	// No source in this machine yet - see the header.
	_StarvedUpstream : BOOL;
	_BlockedDownstream : BOOL;
	_LowMaterial : BOOL;
	_MaterialExhausted : BOOL;

	// One flash clock for the whole indication system. The panel's button lamps
	// read it back through the module so every flashing lamp blinks in phase.
	_FlashTime : TIME := T#500MS;
	_Flash : BOOL;
	FlashTimer : TON;

	RedFlash : BOOL;
	RedSolid : BOOL;
	AmberFlash : BOOL;
	AmberSolid : BOOL;
	BlueFlash : BOOL;
	BlueSolid : BOOL;
	GreenFlash : BOOL;
	GreenSolid : BOOL;

	// Signal tower - the four lamps as driven, and the conditions behind them
	{ attribute 'TcHmiSymbol.AddSymbol' }
	HMI : ST_SignalTower_HMI;
END_VAR

// Amber solid. No source in this machine yet.
PROPERTY BlockedDownstream : BOOL
GET
BlockedDownstream := _BlockedDownstream;
END_GET
SET
_BlockedDownstream := BlockedDownstream;
END_SET
END_PROPERTY

METHOD PUBLIC CyclicLogic
VAR_INPUT
END_VAR
IF NOT _InitComplete THEN
	_InitComplete := Initialize();
	RETURN;
END_IF

// --- Flash clock ------------------------------------------------------------
// Self-retriggering TON. One clock for every flashing lamp on the machine.
FlashTimer(IN := NOT FlashTimer.Q, PT := _FlashTime);
IF FlashTimer.Q THEN
	_Flash := NOT _Flash;
END_IF

// --- Red: Abnormal Stop (flash) / Controlled Stop (solid) -------------------
RedFlash :=	(_State = Tc3_PackML_V2.E_PMLState.ePMLState_Aborting)
		OR	(_State = Tc3_PackML_V2.E_PMLState.ePMLState_Clearing)
		OR	(_State = Tc3_PackML_V2.E_PMLState.ePMLState_Aborted);

RedSolid :=	(_State = Tc3_PackML_V2.E_PMLState.ePMLState_Complete)
		OR	(_State = Tc3_PackML_V2.E_PMLState.ePMLState_Stopped)
		OR	(_State = Tc3_PackML_V2.E_PMLState.ePMLState_Stopping)
		OR	(_State = Tc3_PackML_V2.E_PMLState.ePMLState_Resetting);

// --- Amber: Starved Upstream (flash) / Blocked Downstream (solid) -----------
AmberFlash := _StarvedUpstream AND
			((_State = Tc3_PackML_V2.E_PMLState.ePMLState_Suspending)
		OR	 (_State = Tc3_PackML_V2.E_PMLState.ePMLState_Suspended));

AmberSolid := _BlockedDownstream AND
			((_State = Tc3_PackML_V2.E_PMLState.ePMLState_Suspending)
		OR	 (_State = Tc3_PackML_V2.E_PMLState.ePMLState_Suspended));

// --- Blue: Low Material (flash) / Material Exhausted (solid) ----------------
// Low Material flashes in every state EXCEPT Holding and Held, which is where
// Material Exhausted takes the lamp solid instead.
BlueFlash := _LowMaterial AND
		NOT	((_State = Tc3_PackML_V2.E_PMLState.ePMLState_Holding)
		OR	 (_State = Tc3_PackML_V2.E_PMLState.ePMLState_Held));

BlueSolid := _MaterialExhausted AND
			((_State = Tc3_PackML_V2.E_PMLState.ePMLState_Holding)
		OR	 (_State = Tc3_PackML_V2.E_PMLState.ePMLState_Held));

// --- Green: Ready to Start (flash) / Running (solid) ------------------------
GreenFlash := (_State = Tc3_PackML_V2.E_PMLState.ePMLState_Idle);

GreenSolid :=	(_State = Tc3_PackML_V2.E_PMLState.ePMLState_Starting)
			OR	(_State = Tc3_PackML_V2.E_PMLState.ePMLState_Execute)
			OR	(_State = Tc3_PackML_V2.E_PMLState.ePMLState_Completing)
			OR	(_State = Tc3_PackML_V2.E_PMLState.ePMLState_Unholding)
			OR	(_State = Tc3_PackML_V2.E_PMLState.ePMLState_Unsuspending);

// --- Drive the lamps --------------------------------------------------------
Red	:= (RedFlash	AND _Flash) OR RedSolid;
Yellow	:= (AmberFlash	AND _Flash) OR AmberSolid;
Blue	:= (BlueFlash	AND _Flash) OR BlueSolid;
Green	:= (GreenFlash	AND _Flash) OR GreenSolid;

_Busy	:= FALSE;
_Error	:= FALSE;

SUPER^.CyclicLogic();

// Device config and status only; the inherited half is bridged in
// HMICommunication. The lamps are published ALREADY BLENDED - a flashing lamp
// reads TRUE/FALSE at the flash rate - so a panel bound to these mirrors the
// real tower instead of re-deriving the state table and drifting from it.
HMI.DeviceConfig.FlashTime		:= _FlashTime;
HMI.Device.Red					:= Red;
HMI.Device.Yellow				:= Yellow;
HMI.Device.Blue					:= Blue;
HMI.Device.Green				:= Green;
HMI.Device.Flash				:= _Flash;
HMI.Device.StarvedUpstream		:= _StarvedUpstream;
HMI.Device.BlockedDownstream	:= _BlockedDownstream;
HMI.Device.LowMaterial			:= _LowMaterial;
HMI.Device.MaterialExhausted	:= _MaterialExhausted;
END_METHOD

METHOD PROTECTED HMICommunication
VAR_INPUT
END_VAR
// HMI is a published mirror of the base's own ComponentBase_HMI - carry operator
// intent in before the base looks, and its answers back out afterwards.
ComponentBase_HMI.Command := HMI.Command;

SUPER^.HMICommunication();

HMI.Config	:= ComponentBase_HMI.Config;
HMI.Status	:= ComponentBase_HMI.Status;
HMI.Command	:= ComponentBase_HMI.Command;

// A zero flash time would stop the clock dead and leave every flashing lamp
// stuck on whichever half it was in, so it is refused rather than obeyed.
IF HMI.DeviceConfig.FlashTime > T#0S THEN
	_FlashTime := HMI.DeviceConfig.FlashTime;
END_IF
END_METHOD

// The shared flash phase, so the panel's button lamps blink with the tower.
PROPERTY Flash : BOOL
GET
Flash := _Flash;
END_GET
END_PROPERTY

// Half period of the flash clock.
PROPERTY FlashTime : TIME
GET
FlashTime := _FlashTime;
END_GET
SET
_FlashTime := FlashTime;
END_SET
END_PROPERTY

METHOD PROTECTED Initialize : BOOL
VAR_INPUT
END_VAR
Initialize := SUPER^.Initialize();
END_METHOD

// Blue flashing. No source in this machine yet.
PROPERTY LowMaterial : BOOL
GET
LowMaterial := _LowMaterial;
END_GET
SET
_LowMaterial := LowMaterial;
END_SET
END_PROPERTY

// Blue solid. No source in this machine yet.
PROPERTY MaterialExhausted : BOOL
GET
MaterialExhausted := _MaterialExhausted;
END_GET
SET
_MaterialExhausted := MaterialExhausted;
END_SET
END_PROPERTY

// Amber flashing. No source in this machine yet.
PROPERTY StarvedUpstream : BOOL
GET
StarvedUpstream := _StarvedUpstream;
END_GET
SET
_StarvedUpstream := StarvedUpstream;
END_SET
END_PROPERTY

// The MACHINE's PackML state, written down by the owning module every scan.
PROPERTY State : Tc3_PackML_V2.E_PMLState
GET
State := _State;
END_GET
SET
_State := State;
END_SET
END_PROPERTY

END_FUNCTION_BLOCK

// ---- Library/POUs/F_PMLStateName.TcPOU
// The PackML state as text, for an HMI to display directly.
// IN THE PLC, NOT THE PANEL: tchmiconfig.json sets binding.symbolError to
// "Ignore", so a client-side enum conversion that fails to resolve renders an
// empty control and reports nothing, anywhere.
// Names are the Tc3_PackML_V2 members with the ePMLState_ prefix dropped.
FUNCTION F_PMLStateName : STRING(20)
VAR_INPUT
	State	: E_PMLState;
END_VAR

CASE State OF
	E_PMLState.ePMLState_Clearing:		F_PMLStateName := 'Clearing';
	E_PMLState.ePMLState_Stopped:		F_PMLStateName := 'Stopped';
	E_PMLState.ePMLState_Starting:		F_PMLStateName := 'Starting';
	E_PMLState.ePMLState_Idle:			F_PMLStateName := 'Idle';
	E_PMLState.ePMLState_Suspended:		F_PMLStateName := 'Suspended';
	E_PMLState.ePMLState_Execute:		F_PMLStateName := 'Execute';
	E_PMLState.ePMLState_Stopping:		F_PMLStateName := 'Stopping';
	E_PMLState.ePMLState_Aborting:		F_PMLStateName := 'Aborting';
	E_PMLState.ePMLState_Aborted:		F_PMLStateName := 'Aborted';
	E_PMLState.ePMLState_Holding:		F_PMLStateName := 'Holding';
	E_PMLState.ePMLState_Held:			F_PMLStateName := 'Held';
	E_PMLState.ePMLState_Unholding:		F_PMLStateName := 'Unholding';
	E_PMLState.ePMLState_Suspending:	F_PMLStateName := 'Suspending';
	E_PMLState.ePMLState_Unsuspending:	F_PMLStateName := 'Unsuspending';
	E_PMLState.ePMLState_Resetting:		F_PMLStateName := 'Resetting';
	E_PMLState.ePMLState_Completing:	F_PMLStateName := 'Completing';
	E_PMLState.ePMLState_Complete:		F_PMLStateName := 'Complete';
ELSE
	// ePMLState_Undefined, and anything a future library version adds.
	F_PMLStateName := 'Undefined';
END_CASE

END_FUNCTION

// ---- Modules/10 FG_Transport/FG_Transport.TcPOU
// FG_Transport - two level pallet conveyor, Bosch TS style, closed ring.
// Eleven stations: 5 Index, 4 Stopper, 2 Lift, plus the two main conveyors,
// which are the only thing this level owns itself.
// WireRing is the ONLY place the chain order exists - no station knows what
// follows it, which is what lets one FB serve five index units.
// Contract: _workflow/reference/transport-behaviour.md
FUNCTION_BLOCK FG_Transport EXTENDS FB_PackML_BaseModule
VAR	
	Index01			: FB_TransferIndex := (Name := 'Index01');
	Index02			: FB_TransferIndex := (Name := 'Index02');
	Index03			: FB_TransferIndex := (Name := 'Index03');
	Index04			: FB_TransferIndex := (Name := 'Index04');
	Index05			: FB_TransferIndex := (Name := 'Index05');
	Stopper01		: FB_TransferStopper := (Name := 'Stopper01');
	Stopper02		: FB_TransferStopper := (Name := 'Stopper02');
	Stopper03		: FB_TransferStopper := (Name := 'Stopper03');
	Stopper04		: FB_TransferStopper := (Name := 'Stopper04');
	Lift01			: FB_TransferLift := (Name := 'Lift01');
	Lift02			: FB_TransferLift := (Name := 'Lift02');
	Transport01		: FB_AbstractBinaryDrive := (Name := 'Transport01');
	Transport02		: FB_AbstractBinaryDrive := (Name := 'Transport02');
	
	{ attribute 'TcHmiSymbol.AddSymbol' }
	HMI : ST_BaseModule_HMI;
END_VAR

METHOD PROTECTED Aborting
VAR_INPUT
END_VAR
CASE SequenceState OF
	0:
		NoStateTasksToComplete	:= FALSE;
		Transport01.RunForward := FALSE;
		Transport01.RunBackward := FALSE;
		Transport02.RunForward := FALSE;
		Transport02.RunBackward := FALSE;
		SequenceState			:= SequenceState + 10;

	10:
		StateTasksComplete := TRUE;
END_CASE

SUPER^.Aborting();
END_METHOD

METHOD PROTECTED Clearing
VAR_INPUT
END_VAR
CASE SequenceState OF
	0:
		NoStateTasksToComplete := FALSE;
		SequenceState := SequenceState + 10;

	10:
		IF Transport01.Reset() AND Transport02.Reset() THEN
			StateTasksComplete := TRUE;
		END_IF
END_CASE

SUPER^.Clearing();
END_METHOD

METHOD PUBLIC CyclicLogic
VAR_INPUT
END_VAR
IF NOT _InitComplete THEN
	_InitComplete := Initialize();
	RETURN;
END_IF

// Ring wiring, then the state machine. There is no process image step: every
// component owns its hardware variables and is linked to a terminal channel by
// the imported Mapping_PLC.xml, not by anything in this file.
//
// The chain order lives here and nowhere else - no sub module knows which unit
// follows it. Done before the state machine so a unit sees this scan's values.
WireRing();

// Components get no PackML state callbacks, so the owning module removes every run
// request outside the states entitled to drive them.
// TWO STATES DRIVE THE CONVEYORS: Execute, and Resetting - which runs them to
// accumulate loose pallets against the blocking stoppers.
// THIS GUARD RUNS BEFORE SUPER^.CyclicLogic(), so it does not merely veto the
// output for a scan - it ERASES the request the state method set on the previous
// scan. A state left out of this condition cannot move a conveyor at all,
// however plainly its own code commands one.
IF (_CurrentState <> E_PMLState.ePMLState_Execute)
	AND (_CurrentState <> E_PMLState.ePMLState_Resetting) THEN
	Transport01.RunForward := FALSE;
	Transport01.RunBackward := FALSE;
	Transport02.RunForward := FALSE;
	Transport02.RunBackward := FALSE;
END_IF

SUPER^.CyclicLogic();

PublishStatus();
END_METHOD

METHOD PROTECTED Execute
VAR_INPUT
END_VAR
// The stations sequence themselves - SUPER^.Execute() drives all eleven sub
// modules' Execute methods. This level only owns what belongs to no station:
// the two main conveyors.
//
// There is no step chain here and no completion. A transport ring runs until it
// is stopped, so Execute never calls Complete.

CASE _CurrentMode OF

	//============================= PRODUCTION =================================
	E_PMLUnitMode.ePMLUnitMode_Production:		
		Transport01.RunBackward := TRUE;
		Transport02.RunBackward := TRUE;
		Transport01.RunForward  := FALSE;
		Transport02.RunForward  := FALSE;

	//======================= MAINTENANCE & MANUAL =============================
	E_PMLUnitMode.ePMLUnitMode_Maintenance, E_PMLUnitMode.ePMLUnitMode_Manual:
		// Nothing to do at this level. Each drive honours its own
		// HMI.DeviceCommand struct in these modes - see
		// FB_AbstractBinaryDrive.HMICommunication - so a panel talks to the
		// device it is pointing at rather than through a group GVL. The eleven
		// stations' cylinders do the same through their SPT SolenoidHMI structs.
		;
END_CASE

SUPER^.Execute();
END_METHOD

METHOD PROTECTED HMICommunication
VAR_INPUT
END_VAR
// The command half of the HMI bridge; PublishStatus is the status half.
//
// Without this, the group's published Command block is decoration: the base reads
// its own PackMLBaseModule_HMI.Command and never looks at ours, so a mode or state
// button on the FG_Transport tile would write into a struct nothing consumes.
// It has to happen here because the base calls this method immediately before
// ModeControl() and StateControl().
PackMLBaseModule_HMI.Command := HMI.Command;

SUPER^.HMICommunication();

// The base clears a latch by writing back the value it acted on.
HMI.Command := PackMLBaseModule_HMI.Command;
END_METHOD

METHOD PROTECTED Initialize : BOOL;
VAR
END_VAR
Initialize := FALSE;

CASE DescendantSequenceState OF
	0:
		// HMI.Config.Name is NOT set here. The SPT base writes Config.Name from
		// _Name every scan in its own HMICommunication, and PublishStatus copies
		// the whole Config across - setting it here would be a second author for
		// one field and the first to drift.

		// Eleven station submodules plus two drive components. Forgetting one is
		// silent: its cyclic framework logic would simply never be called.
		RegisterSubmodule(Index01);
		RegisterSubmodule(Index02);
		RegisterSubmodule(Index03);
		RegisterSubmodule(Index04);
		RegisterSubmodule(Index05);
		RegisterSubmodule(Stopper01);
		RegisterSubmodule(Stopper02);
		RegisterSubmodule(Stopper03);
		RegisterSubmodule(Stopper04);
		RegisterSubmodule(Lift01);
		RegisterSubmodule(Lift02);
		RegisterComponent(Transport01);
		RegisterComponent(Transport02);

		// Devices that belong to the group rather than to a station.
		_LogModeChanges		:= FALSE;
		_LogStateChanges	:= TRUE;
		DescendantSequenceState := DescendantSequenceState + 10;

	10:
		// Lift01 raises: it loads at the retracted (lower) end.
		// Lift02 lowers: the mirror image. This one parameter is the entire
		// difference between the two instances.
		Lift01.ReverseDirection := FALSE;
		Lift02.ReverseDirection := TRUE;

		DescendantSequenceState := DescendantSequenceState + 10;

	20:
		IF SUPER^.Initialize() THEN
			DescendantSequenceState := DescendantSequenceState + 10;
		END_IF

	30:
		Initialize := TRUE;
END_CASE
END_METHOD

// TRUE while index unit <Index> is holding a pallet stopped and lifted, waiting
// for its functional group to run. The Machine module polls this and turns it
// into a Start command on the matching group.
//
// A method rather than five properties so the caller can loop 1..5.
METHOD PUBLIC IsIndexReadyForOperation : BOOL
VAR_INPUT
	Index : INT;	// 1..5
END_VAR
CASE Index OF
	1:	IsIndexReadyForOperation := Index01.ReadyForOperation;
	2:	IsIndexReadyForOperation := Index02.ReadyForOperation;
	3:	IsIndexReadyForOperation := Index03.ReadyForOperation;
	4:	IsIndexReadyForOperation := Index04.ReadyForOperation;
	5:	IsIndexReadyForOperation := Index05.ReadyForOperation;
ELSE
	IsIndexReadyForOperation := FALSE;
END_CASE
END_METHOD

ACTION PublishStatus:
// The status half of the HMI bridge; HMICommunication is the command half.
//
// Called from CyclicLogic AFTER SUPER^.CyclicLogic(), so everything below is this
// scan's value. The three fields this action used to set by hand - Mode, State and
// the step index - were the only three that were ever current; Busy, Error,
// ErrorID and HMIControlAvailable stayed at zero because nothing wrote them.
// Copying the base's struct wholesale fixes that and cannot drift.
HMI.Config		:= PackMLBaseModule_HMI.Config;
HMI.Status		:= PackMLBaseModule_HMI.Status;

HMI.StateName			:= F_PMLStateName(_CurrentState);
HMI.Sequence.StepIndex	:= SequenceState;
END_ACTION

METHOD PROTECTED Resetting
VAR_INPUT
END_VAR
// Every station homes itself through its own Resetting, reached by SUPER^.
// This level owns what belongs to no station: the two main conveyors.
// THE CONVEYORS RUN DURING THE RESET, in the production direction. Safe because
// nothing opens: a stopper blocks and is never released, an index blocks before
// lowering. Loose pallets accumulate against the blocking stoppers where a detect
// sensor can see them. It is also what lets a lift hand on a pallet it was
// carrying when it was interrupted, instead of pushing it onto a dead belt.

CASE SequenceState OF
	0:
		NoStateTasksToComplete	:= FALSE;
		Transport01.RunBackward := TRUE;
		Transport02.RunBackward := TRUE;
		Transport01.RunForward  := FALSE;
		Transport02.RunForward  := FALSE;
		SequenceState			:= SequenceState + 10;

	10:
		// The state does not end here: SUPER^ holds it open until all eleven stations
		// have finished their own Resetting, each ending with a fixed accumulation
		// wait, so the belts run for the whole settling period.
		// THE ACCUMULATION IS THE RESET. Once it has settled, every station's state is
		// simply what its sensor says - which is why nothing here waits on an event
		// that might never arrive.
		StateTasksComplete := TRUE;
END_CASE

SUPER^.Resetting();
END_METHOD

// Reports back to index unit <Index> that its functional group has finished, so
// the pallet may be lowered and released. Written by the Machine module.
//
// The index unit clears the flag itself once it has seen it - the group never has
// to reset anything, which is the contract the twin's SIL establishes.
METHOD PUBLIC SetIndexOperationDone
VAR_INPUT
	Index	: INT;		// 1..5
	Value	: BOOL;
END_VAR
CASE Index OF
	1:	Index01.OperationDone := Value;
	2:	Index02.OperationDone := Value;
	3:	Index03.OperationDone := Value;
	4:	Index04.OperationDone := Value;
	5:	Index05.OperationDone := Value;
END_CASE
END_METHOD

METHOD PROTECTED Stopping
VAR_INPUT
END_VAR
CASE SequenceState OF
	0:
		NoStateTasksToComplete	:= FALSE;
		// The drives are components: they have no state methods of their own, so
		// nothing here reaches them through SUPER^. The guard in CyclicLogic is
		// what stops them, and Stopping is not one of the states it exempts.
		SequenceState			:= SequenceState + 10;

	10:
		StateTasksComplete := TRUE;
END_CASE

SUPER^.Stopping();
END_METHOD

ACTION WireRing:
// The chain, exactly as probed from the scene. This is the only place the order
// is written down; no station knows what follows it, which is what lets one FB
// serve five index units.
//
//   Lift01 -> Stopper03 -> Index01 -> Index02 -> Index03 -> Index04 -> Index05
//          -> Stopper04 -> Lift02 -> Stopper01 -> Stopper02 -> Lift01
//
// THE WIRING IS THE AUTHORITY. Two authored Role entries in the twin name the
// wrong successor - both skip the intervening stopper.

// --- Successor readiness: nobody releases into a station that cannot take it ---
//
// ONE CHANNEL, VALID IN EVERY STATE. CanAccept is a derived property - cylinder
// position, detect sensor, transfer latch, no outstanding fault - so it answers
// the same question during Resetting as during Execute. That is what lets a lift's
// reset recovery hand its pallet over on the ordinary contract instead of needing
// a second, reset-only channel wired alongside this one.
Lift01.NextCanAccept	:= Stopper03.CanAccept;
Stopper03.NextCanAccept	:= Index01.CanAccept;
Index01.NextCanAccept	:= Index02.CanAccept;
Index02.NextCanAccept	:= Index03.CanAccept;
Index03.NextCanAccept	:= Index04.CanAccept;
Index04.NextCanAccept	:= Index05.CanAccept;
Index05.NextCanAccept	:= Stopper04.CanAccept;
Stopper04.NextCanAccept	:= Lift02.CanAccept;
Lift02.NextCanAccept	:= Stopper01.CanAccept;
Stopper01.NextCanAccept	:= Stopper02.CanAccept;
Stopper02.NextCanAccept	:= Lift01.CanAccept;

// --- Payload announcements ---------------------------------------------------
// Only a lift acts on being told a pallet is coming: it reverses its belt to draw
// the pallet aboard. Every other station picks a pallet up on its own detect
// sensor, so the announcement would be inert and is not wired.
//
// A lift is a pulling station; the units it feeds are pushing stations. That
// asymmetry is deliberate, not an oversight - see interfaces.md.
Lift01.PayloadIncoming := Stopper02.SendToNext;
Lift02.PayloadIncoming := Stopper04.SendToNext;
END_ACTION

END_FUNCTION_BLOCK

// ---- Modules/10 FG_Transport/FB_TransferIndex.TcPOU
// Index unit - stops a pallet, lifts it clear, runs its functional group,
// then releases. Five instances; the ring wiring decides which is which.
// CanAccept/Occupied are GETTERS, never stored: a remembered readiness flag
// maintained inside Execute is stale in every other state.
// Contract: _workflow/reference/transport-behaviour.md
FUNCTION_BLOCK FB_TransferIndex EXTENDS FB_PackML_BaseModule
VAR
	// --- Components ---------------------------------------------------------
	{ attribute 'TcHmiSymbol.AddSymbol' }
	B_Detect		: FB_DigitalSensor;
	{ attribute 'TcHmiSymbol.AddSymbol' }
	B_Exit			: FB_DigitalSensor;
	{ attribute 'TcHmiSymbol.AddSymbol' }
	Y_Lift			: FB_DoubleSolenoidFeedback;
	{ attribute 'TcHmiSymbol.AddSymbol' }
	Y_Stopper		: FB_SingleSolenoidFeedback;


	// --- Ring handshake -----------------------------------------------------
	// THE INTERFACE IS DERIVED, NOT ASSIGNED. CanAccept and Occupied are getters,
	// correct in every PackML state and mode. There is no _Ready to go stale.
	// _Transferring is the ONE piece of memory: a payload is crossing right now.
	// Set on commit to release, cleared by a B_Exit EDGE in CyclicLogic so it
	// happens in every state.
	_Transferring	: BOOL;
	// Edge detector for the clearing rule. A LEVEL cannot be used: B_Exit may still
	// be made by the previous pallet at the moment this unit commits to the next
	// release, which would clear the latch instantly. The rising edge after the
	// commit is unambiguous, and unlike a cylinder position it is not erased by
	// Stopping or Aborting.
	ExitEdge		: R_TRIG;
	// The successor can physically accept a pallet. Supplied by the parent.
	_NextCanAccept	: BOOL;

	// --- Functional group handshake -----------------------------------------
	// The group is a sibling equipment module, so the Machine module brokers this:
	// it reads ReadyForOperation, commands the group, and writes OperationDone
	// back. This unit never names a functional group.
	_ReadyForOperation	: BOOL;		// pallet is stopped and lifted - run your operation
	_OperationDone		: BOOL;		// the group reports finished

	// The group is not available: it is switched out, or it does not exist yet.
	// The pallet is still stopped, lifted and fixed exactly as always - only the
	// request to run is skipped, so the station is passed rather than skipped and
	// the ring keeps its timing. Routed in by the Machine module, same as the rest.

	// --- Diagnostics --------------------------------------------------------
	// 0 none  1 no home  2 lift did not raise  3 group did not finish
	// 4 lift did not lower  5 no release  6 pallet never reached the exit sensor
	_FaultCode		: DINT;

	// --- Parameters, set by the parent in Initialize ------------------------
	_BlockTime		: TIME := T#2S;
	_LiftTime		: TIME := T#3S;
	_OperationTime	: TIME := T#60S;	// how long a station may take
	_ReleaseTime	: TIME := T#2S;
	_ClearTime		: TIME := T#10S;
	// How long a reset lets the line settle once this unit is blocking and lowered.
	// The group runs the main conveyors throughout, so pallets travel up against the
	// blocking stoppers and accumulate where a detect sensor can see them.
	_AccumulateTime	: TIME := T#5S;

	// --- HMI ----------------------------------------------------------------
	// One struct for the whole tile, extending the SPT module interface. The
	// inherited half is bridged to the base's own PackMLBaseModule_HMI in two
	// places: HMICommunication pushes Command in before the base acts on it,
	// PublishHMI copies Config and Status back out after. The Station half is this
	// block's own and is filled by PublishHMI alone.
	{ attribute 'TcHmiSymbol.AddSymbol' }
	HMI	: ST_TransferIndex_HMI;
END_VAR

METHOD PROTECTED Aborting
VAR_INPUT
END_VAR
CASE SequenceState OF
	0:
		NoStateTasksToComplete	:= FALSE;
		// Block, and withdraw the request to the station. The lift is left where
		// it is on purpose - dropping a pallet that a station still has hold of
		// is worse than leaving it raised. An abort is immediate by definition, so
		// unlike Resetting it does not wait for a crossing to finish.
		//
		// Nothing else is cleared: the interface is derived, and _Transferring is
		// cleared by B_Exit whenever the pallet actually gets there.
		Y_Stopper.Retract();
		_ReadyForOperation	:= FALSE;
		SequenceState		:= SequenceState + 10;

	10:
		StateTasksComplete := TRUE;
END_CASE

SUPER^.Aborting();
END_METHOD

METHOD PROTECTED Clearing
VAR_INPUT
END_VAR
CASE SequenceState OF
	0:
		NoStateTasksToComplete := FALSE;
		_FaultCode := 0;
		SequenceState := SequenceState + 10;

	10:	// Clear latched component alarms - the lift's travel timeout latches.
		IF Y_Lift.Reset()
			AND Y_Stopper.Reset()
			AND B_Detect.Reset()
			AND B_Exit.Reset() THEN
			SequenceState := SequenceState + 10;
		END_IF

	20:
		StateTasksComplete := TRUE;
END_CASE

SUPER^.Clearing();
END_METHOD

METHOD PUBLIC CyclicLogic
VAR_INPUT
END_VAR
IF NOT _InitComplete THEN
	_InitComplete := Initialize();
	RETURN;
END_IF

// Nothing to copy: every component is linked to its terminal at the instance
// declaration in FG_Transport.

// THE TRANSFER LATCH IS CLEARED BY THE SENSOR, IN EVERY STATE - not in the
// Execute step that starts the release. A pallet that finishes crossing while
// the machine is stopped or resetting has still finished crossing.
//
// THE WITNESS MUST BE A SENSOR EDGE. Qualifying it with Y_Stopper.Extended
// deadlocked the machine: Stopping and Aborting retract the cylinder immediately,
// destroying the very witness the rule depended on. A rising edge is specific to
// THIS crossing and no state change can erase it.
ExitEdge(CLK := B_Exit.Active);
IF _Transferring AND ExitEdge.Q THEN
	_Transferring := FALSE;
END_IF

SUPER^.CyclicLogic();

// After the base, so the published struct carries this scan's state and
// this scan's HMI permission rather than last scan's.
PublishHMI();
END_METHOD

METHOD PROTECTED Execute
VAR_INPUT
END_VAR
VAR_INST
	HomeTimer		: TON;
	LiftUpTimer		: TON;
	OperationTimer	: TON;
	LiftDownTimer	: TON;
	ReleaseTimer	: TON;
	ClearTimer		: TON;
END_VAR
// The ring runs continuously, so this state loops instead of completing.

CASE _CurrentMode OF

	//============================= PRODUCTION =================================
	E_PMLUnitMode.ePMLUnitMode_Production:

		CASE SequenceState OF
			0:	// Home: blocking, lift down, nothing outstanding. The handshake
				// interface is derived and needs nothing cleared here; only the
				// group request, which is this unit's own bookkeeping.
				NoStateTasksToComplete	:= FALSE;
				Y_Stopper.Retract();
				Y_Lift.Retract();
				_ReadyForOperation	:= FALSE;
				_OperationDone		:= FALSE;
				SequenceState		:= SequenceState + 10;

			10:	// Blocking position comes from the real switch; the lift has a
				// genuine feedback component and reports its own position.
				// CanAccept becomes TRUE by itself once both are home and the
				// detect sensor is clear - this unit never publishes readiness, so
				// there is no window in which it advertises it over a pallet.
				IF Y_Stopper.Retracted AND Y_Lift.Retracted THEN
					SequenceState	:= SequenceState + 10;
				ELSIF HomeTimer.Q THEN
					_FaultCode := 1;
					ChangeState(E_PMLCommand.ePMLCommand_Hold);
				END_IF

			20:	// Idle and empty - the normal resting condition
				IF B_Detect.Active THEN
					SequenceState	:= SequenceState + 10;
				END_IF

			30:	// Invariant 1 - lift the pallet clear while the stopper still
				// holds it, and only then let the station run.
				Y_Lift.Extend();
				IF Y_Lift.Extended THEN
					SequenceState	:= SequenceState + 10;
				ELSIF LiftUpTimer.Q THEN
					_FaultCode := 2;
					ChangeState(E_PMLCommand.ePMLCommand_Hold);
				END_IF

			40:	// Ask the group to run and wait for it. The Machine module
				// brokers both halves; this unit clears the done flag itself, so
				// the group never has to reset anything.
				//
				// A group that is not implemented is handled by the broker, which
				// answers SetIndexOperationDone immediately - see
				// Machine.BrokerIndexHandshakes. This unit neither knows nor cares
				// which groups exist.
				_ReadyForOperation := TRUE;
				IF _OperationDone THEN
					_OperationDone		:= FALSE;
					_ReadyForOperation	:= FALSE;
					SequenceState		:= SequenceState + 10;
				ELSIF OperationTimer.Q THEN
					_FaultCode := 3;
					ChangeState(E_PMLCommand.ePMLCommand_Hold);
				END_IF

			50:	// Invariant 2 - the operation is complete, so the lift may drop
				Y_Lift.Retract();
				IF Y_Lift.Retracted THEN
					SequenceState := SequenceState + 10;
				ELSIF LiftDownTimer.Q THEN
					_FaultCode := 4;
					ChangeState(E_PMLCommand.ePMLCommand_Hold);
				END_IF

			60:	// Invariant 3 - the successor can physically accept before release
				IF _NextCanAccept THEN
					// The crossing starts here; cleared by B_Exit in CyclicLogic.
					_Transferring	:= TRUE;
					SequenceState	:= SequenceState + 10;
				END_IF

			70:	// Release
				Y_Stopper.Extend();
				IF Y_Stopper.Extended THEN
					SequenceState := SequenceState + 10;
				ELSIF ReleaseTimer.Q THEN
					_FaultCode := 5;
					ChangeState(E_PMLCommand.ePMLCommand_Hold);
				END_IF

			80:	// Confirm the pallet actually left
				IF B_Exit.Active THEN
					SequenceState := 0;
				ELSIF ClearTimer.Q THEN
					_FaultCode := 6;
					ChangeState(E_PMLCommand.ePMLCommand_Hold);
				END_IF
		END_CASE

	//======================= MAINTENANCE & MANUAL =============================
	E_PMLUnitMode.ePMLUnitMode_Maintenance, E_PMLUnitMode.ePMLUnitMode_Manual:
		// Both cylinders are SPT components and honour their own SolenoidHMI
		// structs whenever the mode grants HMI control. The handshake interface is
		// derived from the sensors, so it keeps telling the truth while an operator
		// moves pallets by hand; only the group request is withdrawn.
		_ReadyForOperation	:= FALSE;
END_CASE

SUPER^.Execute();

HomeTimer(		IN := (SequenceState = 10),							PT := _BlockTime);
LiftUpTimer(	IN := (SequenceState = 30),							PT := _LiftTime);
OperationTimer(	IN := (SequenceState = 40),							PT := _OperationTime);
LiftDownTimer(	IN := (SequenceState = 50),							PT := _LiftTime);
ReleaseTimer(	IN := (SequenceState = 70),							PT := _ReleaseTime);
ClearTimer(		IN := (SequenceState = 80),							PT := _ClearTime);
END_METHOD

// 0 none  1 no home  2 lift did not raise  3 group did not finish
// 4 lift did not lower  5 no release  6 pallet never reached the exit sensor
PROPERTY FaultCode : DINT
GET
FaultCode := _FaultCode;
END_GET
END_PROPERTY

METHOD PROTECTED HMICommunication
VAR_INPUT
END_VAR
// The command half of the HMI bridge. The status half is PublishHMI.
// MUST be in this method, not in PublishHMI. The base calls it immediately before
// ModeControl() and StateControl(), and reads its OWN PackMLBaseModule_HMI.Command,
// never ours. A command written after SUPER^.CyclicLogic() returns is a full scan
// too late, every time.
PackMLBaseModule_HMI.Command := HMI.Command;

SUPER^.HMICommunication();

// The base clears a command latch by writing the value it acted on back into
// Command.Mode / Command.State. Carry that back out so the panel sees its request
// consumed rather than re-issuing it on the next scan.
HMI.Command := PackMLBaseModule_HMI.Command;
END_METHOD

METHOD PROTECTED Initialize : BOOL;
VAR
END_VAR
Initialize := FALSE;

CASE DescendantSequenceState OF
	0:
		RegisterComponent(B_Detect);
		RegisterComponent(B_Exit);
		RegisterComponent(Y_Lift);
		RegisterComponent(Y_Stopper);

		_LogModeChanges		:= FALSE;
		_LogStateChanges	:= FALSE;
		DescendantSequenceState := DescendantSequenceState + 10;

	10:
		// Travel timeouts in ms (LREAL). The lift has real feedback so these
		// alarm on a jam; the stopper is open loop and these only bound the move.
		Y_Lift.ExtendTime		:= 3000.0;
		Y_Lift.RetractTime		:= 3000.0;
		Y_Stopper.ExtendTime	:= 2000.0;
		Y_Stopper.RetractTime	:= 2000.0;
		DescendantSequenceState := DescendantSequenceState + 10;

	20:
		IF SUPER^.Initialize() THEN
			DescendantSequenceState := DescendantSequenceState + 10;
		END_IF

	30:
		Initialize := TRUE;
END_CASE
END_METHOD

// The successor's CanAccept, wired in by the parent.
PROPERTY NextCanAccept : BOOL
SET
_NextCanAccept := NextCanAccept;
END_SET
END_PROPERTY

// This station is physically holding or handling a pallet.
//
// Derived, like CanAccept: the detect sensor, or a crossing that has been committed
// to and not yet confirmed finished. There is no remembered occupancy behind it, so
// there is nothing for a state change or a program download to falsify.
PROPERTY Occupied : BOOL
GET
Occupied := B_Detect.Active OR _Transferring;
END_GET
END_PROPERTY

// Written TRUE by the Machine module when this unit's functional group reports
// its operation complete. This unit clears it again itself.
PROPERTY OperationDone : BOOL
SET
_OperationDone := OperationDone;
END_SET
END_PROPERTY

ACTION PublishHMI:
// Everything an operator tile needs from this unit, in one struct.
//
// Called from CyclicLogic AFTER SUPER^.CyclicLogic(), so _CurrentState and the
// base's HMIControlAvailable are this scan's values and not last scan's.

// --- Inherited half ---------------------------------------------------------
// Straight copies of the struct the SPT base maintains. Nothing is recomputed -
// a second calculation would be a second answer.
// HMIControlAvailable is the gate for every jog button on the tile, and only
// ePMLUnitMode_Manual grants it. Bind button enablement to THIS, not to a
// group-level flag computed as Manual OR Maintenance, which over-reports.
HMI.Config		:= PackMLBaseModule_HMI.Config;
HMI.Status		:= PackMLBaseModule_HMI.Status;

HMI.StateName			:= F_PMLStateName(_CurrentState);
HMI.Sequence.StepIndex	:= SequenceState;

// --- Ring handshake ---------------------------------------------------------
// The derived properties, not backing variables - the tile shows what the machine
// physically is, which is the same thing the neighbouring stations act on. The
// struct field names are unchanged so the existing panel bindings still resolve.
HMI.Station.Ready					:= CanAccept;
HMI.Station.Occupied				:= Occupied;
HMI.Station.NextReady				:= _NextCanAccept;
HMI.Station.SendToNext				:= SendToNext;

// --- Functional group handshake ---------------------------------------------
HMI.Station.ReadyForOperation		:= _ReadyForOperation;
HMI.Station.OperationDone			:= _OperationDone;

// --- Diagnostics ------------------------------------------------------------
HMI.Station.FaultCode				:= _FaultCode;
END_ACTION

// This station can physically take a pallet right now. The predecessor gates its
// release on this, and it is the whole of the readiness contract.
//
// DERIVED, NOT ASSIGNED. Computed from both cylinder limit switches, the detect
// sensor and the transfer latch, so it is correct in every PackML state and every
// mode. The old _Ready was written only inside the Execute step chain, which made
// it stale or FALSE everywhere else.
PROPERTY CanAccept : BOOL
GET
CanAccept := Y_Stopper.Retracted
	AND Y_Lift.Retracted
	AND NOT B_Detect.Active
	AND NOT _Transferring
	AND (_FaultCode = 0);
END_GET
END_PROPERTY

// The pallet is stopped and lifted. The Machine module turns this into a Start
// command on the matching functional group.
PROPERTY ReadyForOperation : BOOL
GET
ReadyForOperation := _ReadyForOperation;
END_GET
END_PROPERTY

METHOD PROTECTED Resetting
VAR_INPUT
END_VAR
VAR_INST
	ResetBlockTimer	: TON;
	ResetLiftTimer	: TON;
	AccumulateTimer	: TON;
END_VAR
// A RESET RE-ESTABLISHES WHERE THE PALLETS ARE.
// Block, drop the lift, then wait for the line to settle. The group runs the main
// conveyors throughout a reset, so whatever was moving accumulates against the
// blocking stoppers; after that each station's state is what its sensor says.
//
// A FIXED WAIT, NOT AN EVENT. Waiting for the in-flight pallet to clear B_Exit
// deadlocked: Stopping had already retracted the cylinder the clearing rule
// needed. A RESET MUST ALWAYS TERMINATE - nothing in it may wait on an event that
// might not arrive.

CASE SequenceState OF
	0:
		NoStateTasksToComplete	:= FALSE;
		Y_Stopper.Retract();
		_ReadyForOperation	:= FALSE;
		_OperationDone		:= FALSE;
		// The routed inputs are not cleared here: they are rewritten every scan by the
		// Machine, and a reset is not the operator changing their mind about it.
		SequenceState		:= SequenceState + 10;

	10:	// Drop the lift only once the stopper is confirmed blocking
		IF Y_Stopper.Retracted THEN
			SequenceState := SequenceState + 10;
		ELSIF ResetBlockTimer.Q THEN
			_FaultCode := 1;
			ChangeState(E_PMLCommand.ePMLCommand_Hold);
		END_IF

	20:
		Y_Lift.Retract();
		IF Y_Lift.Retracted THEN
			SequenceState := SequenceState + 10;
		ELSIF ResetLiftTimer.Q THEN
			_FaultCode := 4;
			ChangeState(E_PMLCommand.ePMLCommand_Hold);
		END_IF

	30:	// Accumulation. When it expires the pallets have settled, so any crossing
		// this unit had outstanding is over by definition. Clearing the latch here
		// is the reset re-establishing state rather than inheriting a crossing whose
		// sensor edge was missed while the machine was stopped.
		IF AccumulateTimer.Q THEN
			_Transferring	:= FALSE;
			SequenceState	:= SequenceState + 10;
		END_IF

	40:
		StateTasksComplete := TRUE;
END_CASE

SUPER^.Resetting();

ResetBlockTimer(IN := (SequenceState = 10),							PT := _BlockTime);
ResetLiftTimer(	IN := (SequenceState = 20),							PT := _LiftTime);
AccumulateTimer(IN := (SequenceState = 30),							PT := _AccumulateTime);
END_METHOD

// This unit is handing a pallet over right now; only a lift acts on it.
//
// This is the transfer latch itself, not a second flag that shadows it. Handing
// over and being mid-crossing are the same fact, so keeping them as one variable
// means they cannot disagree. Cleared by B_Exit.
PROPERTY SendToNext : BOOL
GET
SendToNext := _Transferring;
END_GET
END_PROPERTY

METHOD PROTECTED Stopping
VAR_INPUT
END_VAR
// A controlled stop blocks and withdraws the station request, but leaves the
// lift alone so a part being worked on is not dropped mid-operation.

CASE SequenceState OF
	0:
		NoStateTasksToComplete	:= FALSE;
		// Block and withdraw the station request. Nothing to clear - see Aborting.
		Y_Stopper.Retract();
		_ReadyForOperation	:= FALSE;
		SequenceState		:= SequenceState + 10;

	10:
		StateTasksComplete := TRUE;
END_CASE

SUPER^.Stopping();
END_METHOD

END_FUNCTION_BLOCK

// ---- Modules/10 FG_Transport/FB_TransferStopper.TcPOU
// Accumulation stopper - one pallet, held until the next station is free.
// RETRACTED (min) HOLDS THE PALLET; EXTENDING (max) RELEASES IT. Nine authored
// Function entries in the twin once said the opposite.
// CanAccept/Occupied are GETTERS, never stored.
// Contract: _workflow/reference/transport-behaviour.md
FUNCTION_BLOCK FB_TransferStopper EXTENDS FB_PackML_BaseModule
VAR
	// --- Components ---------------------------------------------------------
	{ attribute 'TcHmiSymbol.AddSymbol' }
	B_Detect		: FB_DigitalSensor;
	{ attribute 'TcHmiSymbol.AddSymbol' }
	B_Exit			: FB_DigitalSensor;
	{ attribute 'TcHmiSymbol.AddSymbol' }
	Y_Stopper		: FB_SingleSolenoidFeedback;


	// --- Ring handshake -----------------------------------------------------
	// THE INTERFACE IS DERIVED, NOT ASSIGNED. CanAccept and Occupied are getters,
	// correct in every PackML state and mode. There is no _Ready to go stale.
	// _Transferring is the ONE piece of memory: a payload is crossing right now.
	// Set on commit to release, cleared by a B_Exit EDGE in CyclicLogic so it
	// happens in every state. A plain BOOL initialising FALSE is the point - a
	// stale FALSE is corrected by B_Detect on the next scan.
	_Transferring	: BOOL;
	// Edge detector for the clearing rule. A LEVEL cannot be used: B_Exit may still
	// be made by the previous pallet at the moment this unit commits to the next
	// release, which would clear the latch instantly. The rising edge after the
	// commit is unambiguous, and unlike a cylinder position or a drive command it
	// is not erased by Stopping or Aborting.
	ExitEdge		: R_TRIG;
	// The successor can physically accept a pallet. Supplied by the parent.
	_NextCanAccept	: BOOL;

	// --- Diagnostics --------------------------------------------------------

	// Module level fault. The SPT components raise their own alarms through the
	// event logger; these codes cover the sequence timeouts, which belong to the
	// unit rather than to any one device. Published for the HMI.
	// 0 none  1 no block  2 no release  3 pallet never reached the exit sensor
	_FaultCode		: DINT;

	// --- Parameters, set by the parent in Initialize ------------------------
	_BlockTime		: TIME := T#2S;		// stopper travel to the blocking position
	_ReleaseTime	: TIME := T#2S;		// stopper travel to the release position
	_ClearTime		: TIME := T#10S;	// pallet to reach the exit sensor once released
	// How long a reset lets the line settle once this unit is blocking. The group
	// runs the main conveyors throughout, so pallets travel up against the blocking
	// stoppers and accumulate where a detect sensor can see them.
	_AccumulateTime	: TIME := T#5S;

	// --- HMI ----------------------------------------------------------------
	// One struct for the whole tile, extending the SPT module interface. The
	// inherited half is bridged to the base's own PackMLBaseModule_HMI in two
	// places: HMICommunication pushes Command in before the base acts on it,
	// PublishHMI copies Config and Status back out after. The Station half is this
	// block's own and is filled by PublishHMI alone.
	{ attribute 'TcHmiSymbol.AddSymbol' }
	HMI	: ST_TransferStopper_HMI;
END_VAR

METHOD PROTECTED Aborting
VAR_INPUT
END_VAR
CASE SequenceState OF
	0:
		NoStateTasksToComplete	:= FALSE;
		// Block on abort. A released stopper would let an unsupervised pallet run
		// into a station that is no longer sequencing. An abort is immediate by
		// definition, so unlike Resetting it does not wait for a crossing to
		// finish - that is the difference between stopping safely and stopping now.
		//
		// Nothing is cleared: the interface is derived, and _Transferring is
		// cleared by B_Exit whenever the pallet actually gets there.
		Y_Stopper.Retract();
		SequenceState	:= SequenceState + 10;

	10:
		StateTasksComplete := TRUE;
END_CASE

SUPER^.Aborting();
END_METHOD

METHOD PROTECTED Clearing
VAR_INPUT
END_VAR
CASE SequenceState OF
	0:
		NoStateTasksToComplete := FALSE;
		_FaultCode := 0;
		SequenceState := SequenceState + 10;

	10:	// Clear latched component alarms.
		IF Y_Stopper.Reset()
			AND B_Detect.Reset()
			AND B_Exit.Reset() THEN
			SequenceState := SequenceState + 10;
		END_IF

	20:
		StateTasksComplete := TRUE;
END_CASE

SUPER^.Clearing();
END_METHOD

METHOD PUBLIC CyclicLogic
VAR_INPUT
END_VAR
IF NOT _InitComplete THEN
	_InitComplete := Initialize();
	RETURN;
END_IF

// No ReadInputs / WriteOutputs anywhere in this group: each component is linked
// to its terminal channel at the instance declaration, so there is no image to
// copy in or out.

// THE TRANSFER LATCH IS CLEARED BY THE SENSOR, IN EVERY STATE - not in the
// Execute step that starts the release. A pallet that finishes crossing while the
// machine is stopped or resetting has still finished crossing.
//
// THE WITNESS MUST BE A SENSOR EDGE. Qualifying it with Y_Stopper.Extended
// deadlocked the machine: Stopping and Aborting retract the cylinder immediately,
// destroying the very witness the rule depended on, so _Transferring could never
// go FALSE again. A rising edge is specific to THIS crossing and no state change
// can erase it.
ExitEdge(CLK := B_Exit.Active);
IF _Transferring AND ExitEdge.Q THEN
	_Transferring := FALSE;
END_IF

SUPER^.CyclicLogic();

// After the base, so the published struct carries this scan's state and
// this scan's HMI permission rather than last scan's.
PublishHMI();
END_METHOD

METHOD PROTECTED Execute
VAR_INPUT
END_VAR
VAR_INST
	BlockTimer		: TON;
	ReleaseTimer	: TON;
	ClearTimer		: TON;
END_VAR
// The transport ring runs continuously, so this state loops rather than
// completing. Execute is the one acting state that does not self-complete and
// SequenceState is simply reset to 0 after each pallet.

CASE _CurrentMode OF

	//============================= PRODUCTION =================================
	E_PMLUnitMode.ePMLUnitMode_Production:

		CASE SequenceState OF
			0:	// Block. Nothing to clear: this chain no longer owns the interface,
				// it only drives the cylinder. CanAccept and Occupied are derived
				// from the sensors and are already correct on entry.
				NoStateTasksToComplete	:= FALSE;
				Y_Stopper.Retract();
				SequenceState	:= SequenceState + 10;

			10:	// Wait for the real limit switch, not the commanded position.
				// CanAccept becomes TRUE by itself the moment the switch makes and
				// the detect sensor is clear - there is no window in which this
				// unit advertises readiness over a pallet, because readiness is
				// not something it publishes.
				IF Y_Stopper.Retracted THEN
					SequenceState	:= SequenceState + 10;
				ELSIF BlockTimer.Q THEN
					_FaultCode := 1;
					ChangeState(E_PMLCommand.ePMLCommand_Hold);
				END_IF

			20:	// Idle and empty. Waiting here is the normal resting condition.
				IF B_Detect.Active THEN
					SequenceState	:= SequenceState + 10;
				END_IF

			30:	// Holding a pallet. Release only onto a successor that can
				// physically accept one - invariant 3.
				IF _NextCanAccept THEN
					// The crossing starts here. This is also what tells a lift to
					// start its belt, so it is set BEFORE the cylinder opens; it is
					// cleared by B_Exit in CyclicLogic, never by this chain.
					_Transferring	:= TRUE;
					SequenceState	:= SequenceState + 10;
				END_IF

			40:	// Release
				Y_Stopper.Extend();
				IF Y_Stopper.Extended THEN
					SequenceState := SequenceState + 10;
				ELSIF ReleaseTimer.Q THEN
					_FaultCode := 2;
					ChangeState(E_PMLCommand.ePMLCommand_Hold);
				END_IF

			50:	// The pallet has to actually leave before this unit takes another.
				// _Transferring has already been cleared by B_Exit in CyclicLogic.
				IF B_Exit.Active THEN
					SequenceState := 0;
				ELSIF ClearTimer.Q THEN
					_FaultCode := 3;
					ChangeState(E_PMLCommand.ePMLCommand_Hold);
				END_IF
		END_CASE

	//======================= MAINTENANCE & MANUAL =============================
	E_PMLUnitMode.ePMLUnitMode_Maintenance, E_PMLUnitMode.ePMLUnitMode_Manual:
		// The stopper is an SPT component and honours its own SolenoidHMI struct
		// whenever the mode grants HMI control. No sequence runs, and nothing needs
		// to be assigned: the interface is derived from the sensors, so it keeps
		// telling the truth while an operator moves pallets by hand.
		;
END_CASE

SUPER^.Execute();

BlockTimer(	IN := (SequenceState = 10),							PT := _BlockTime);
ReleaseTimer(IN := (SequenceState = 40),						PT := _ReleaseTime);
ClearTimer(	IN := (SequenceState = 50),							PT := _ClearTime);
END_METHOD

// Sequence timeout that took this unit to Held. Cleared by Clearing.
// 0 none  1 no block  2 no release  3 pallet never reached the exit sensor
PROPERTY FaultCode : DINT
GET
FaultCode := _FaultCode;
END_GET
END_PROPERTY

METHOD PROTECTED HMICommunication
VAR_INPUT
END_VAR
// The command half of the HMI bridge; PublishHMI is the status half.
// The base calls this immediately before ModeControl() and StateControl(), which
// is the only point at which an operator command can still reach this scan's
// state machine. See FB_TransferIndex.HMICommunication for the full reasoning.
PackMLBaseModule_HMI.Command := HMI.Command;

SUPER^.HMICommunication();

// The base clears a latch by writing back the value it acted on.
HMI.Command := PackMLBaseModule_HMI.Command;
END_METHOD

METHOD PROTECTED Initialize : BOOL;
VAR
END_VAR
Initialize := FALSE;

CASE DescendantSequenceState OF
	0:
		// Names are prefixed by the parent with the unit name, so alarms read
		// "Stopper03 B_Detect" rather than one of four identical "B_Detect".
		RegisterComponent(B_Detect);
		RegisterComponent(B_Exit);
		RegisterComponent(Y_Stopper);

		_LogModeChanges		:= FALSE;
		_LogStateChanges	:= FALSE;
		DescendantSequenceState := DescendantSequenceState + 10;

	10:
		// Open loop travel times. The stopper has no extended limit switch, so
		// these bound the commanded move rather than confirming it.
		Y_Stopper.ExtendTime	:= 2000.0;
		Y_Stopper.RetractTime	:= 2000.0;
		DescendantSequenceState := DescendantSequenceState + 10;

	20:
		IF SUPER^.Initialize() THEN
			DescendantSequenceState := DescendantSequenceState + 10;
		END_IF

	30:
		Initialize := TRUE;
END_CASE
END_METHOD

// The successor's CanAccept, wired in by the parent - this unit does not know the
// chain order.
PROPERTY NextCanAccept : BOOL
SET
_NextCanAccept := NextCanAccept;
END_SET
END_PROPERTY

// This station is physically holding or handling a pallet.
//
// Derived, like CanAccept: the detect sensor, or a crossing that has been committed
// to and not yet confirmed finished. True from the moment the unit decides to
// release until B_Exit says the pallet has gone, which is exactly the window in
// which nobody should send it another one.
//
// There is no remembered occupancy behind this, so there is nothing for a state
// change or a program download to falsify.
PROPERTY Occupied : BOOL
GET
Occupied := B_Detect.Active OR _Transferring;
END_GET
END_PROPERTY

ACTION PublishHMI:
// Everything an operator tile needs from this unit, in one struct.
//
// Called from CyclicLogic AFTER SUPER^.CyclicLogic(), so _CurrentState and the
// base's HMIControlAvailable are this scan's values and not last scan's.

// --- Inherited half ---------------------------------------------------------
// Straight copies of the struct the SPT base maintains - Config carries Name and
// the logging toggles, Status carries Busy, Error, ErrorID, Mode, State and
// HMIControlAvailable. The last is the gate for the jog buttons on the tile,
// granted in ePMLUnitMode_Manual only.
HMI.Config		:= PackMLBaseModule_HMI.Config;
HMI.Status		:= PackMLBaseModule_HMI.Status;

HMI.StateName			:= F_PMLStateName(_CurrentState);
HMI.Sequence.StepIndex	:= SequenceState;

// --- Ring handshake ---------------------------------------------------------
// The derived properties, not backing variables - the tile shows what the machine
// physically is, which is the same thing the neighbouring stations act on. The
// struct field names are unchanged so the existing panel bindings still resolve.
HMI.Station.Ready					:= CanAccept;
HMI.Station.Occupied				:= Occupied;
HMI.Station.NextReady				:= _NextCanAccept;
HMI.Station.SendToNext				:= SendToNext;

// --- Diagnostics ------------------------------------------------------------
HMI.Station.FaultCode				:= _FaultCode;
END_ACTION

// This station can physically take a pallet right now. The predecessor gates its
// release on this, and it is the whole of the readiness contract.
//
// DERIVED, NOT ASSIGNED: computed from the cylinder limit, the detect sensor and
// the transfer latch, so it is correct in every PackML state and mode.
//
// Blocking position, nothing on the sensor, nothing crossing, no fault outstanding.
PROPERTY CanAccept : BOOL
GET
CanAccept := Y_Stopper.Retracted
	AND NOT B_Detect.Active
	AND NOT _Transferring
	AND (_FaultCode = 0);
END_GET
END_PROPERTY

METHOD PROTECTED Resetting
VAR_INPUT
END_VAR
VAR_INST
	ResetBlockTimer	: TON;
	AccumulateTimer	: TON;
END_VAR
// A RESET RE-ESTABLISHES WHERE THE PALLETS ARE.
// Block, then wait for the line to settle. The group runs the main conveyors
// throughout a reset, so whatever was moving accumulates against the blocking
// stoppers; after that, each station's state is simply what its sensor says.
//
// A FIXED WAIT, NOT AN EVENT. Waiting for the in-flight pallet to clear B_Exit
// deadlocked: Stopping had already retracted the cylinder the clearing rule
// needed. A RESET MUST ALWAYS TERMINATE - nothing in it may wait on an event that
// might not arrive.
// The stopper is never released on reset, and is already blocking anyway.

CASE SequenceState OF
	0:
		NoStateTasksToComplete	:= FALSE;
		Y_Stopper.Retract();
		SequenceState	:= SequenceState + 10;

	10:
		IF Y_Stopper.Retracted THEN
			SequenceState := SequenceState + 10;
		ELSIF ResetBlockTimer.Q THEN
			_FaultCode := 1;
			ChangeState(E_PMLCommand.ePMLCommand_Hold);
		END_IF

	20:	// Accumulation. When it expires the pallets have settled, so any crossing
		// this unit had outstanding is over by definition - either the pallet
		// reached the next station or it is back against this one. Clearing the
		// latch here is the reset re-establishing state rather than inheriting a
		// crossing whose sensor edge was missed while the machine was stopped.
		IF AccumulateTimer.Q THEN
			_Transferring	:= FALSE;
			SequenceState	:= SequenceState + 10;
		END_IF

	30:
		StateTasksComplete := TRUE;
END_CASE

SUPER^.Resetting();

ResetBlockTimer(IN := (SequenceState = 10),							PT := _BlockTime);
AccumulateTimer(IN := (SequenceState = 20),							PT := _AccumulateTime);
END_METHOD

// This unit is handing a pallet over right now. The parent forwards it to the
// successor's PayloadIncoming, which only a lift acts on - it starts drawing the
// pallet aboard.
//
// This is the transfer latch itself, not a second flag that shadows it. Handing
// over and being mid-crossing are the same fact, and keeping them as one variable
// means they cannot disagree. It is cleared by B_Exit, so the announcement stops
// exactly when the pallet has actually gone.
PROPERTY SendToNext : BOOL
GET
SendToNext := _Transferring;
END_GET
END_PROPERTY

METHOD PROTECTED Stopping
VAR_INPUT
END_VAR
CASE SequenceState OF
	0:
		NoStateTasksToComplete	:= FALSE;
		// Block. Nothing to clear - see Aborting.
		Y_Stopper.Retract();
		SequenceState	:= SequenceState + 10;

	10:
		StateTasksComplete := TRUE;
END_CASE

SUPER^.Stopping();
END_METHOD

END_FUNCTION_BLOCK

// ---- Modules/10 FG_Transport/FB_TransferLift.TcPOU
// Lift unit - moves a pallet between the two conveyor levels. Two instances.
// THE CARRIAGE BELT MAY ONLY RUN WHILE THE CARRIAGE IS AT A LEVEL; between
// levels it drives the pallet into a fixed edge. Enforced in CyclicLogic for
// every state and mode, including Manual.
// Contract: _workflow/reference/transport-behaviour.md
FUNCTION_BLOCK FB_TransferLift EXTENDS FB_PackML_BaseModule
VAR
	// --- Components ---------------------------------------------------------
	{ attribute 'TcHmiSymbol.AddSymbol' }
	B_Detect		: FB_DigitalSensor;		// on the carriage - pallet is aboard
	{ attribute 'TcHmiSymbol.AddSymbol' }
	B_Exit			: FB_DigitalSensor;		// on the fixed frame - pallet has left
	{ attribute 'TcHmiSymbol.AddSymbol' }
	Y_Lift			: FB_DoubleSolenoidFeedback;

	// --- Carriage belt ------------------------------------------------------
	// A drive module of its own, like the two main conveyor sections, so it can
	// report that it failed to start rather than silently stalling the lift.
	// Backward draws a pallet aboard, forward pushes it off.
	M_Conveyor		: FB_AbstractBinaryDrive := (Name := 'M_Conveyor');

	// --- Ring handshake -----------------------------------------------------
	// THE INTERFACE IS DERIVED, NOT ASSIGNED. CanAccept and Occupied are getters,
	// correct in every PackML state and mode. There is no _Ready to go stale.
	// THE CARRIAGE MUST NOT CHANGE LEVEL while either latch is TRUE - a pallet drawn
	// half aboard has not reached B_Detect, so no sensor can see that case alone.
	// Two BOOLs, not one: the direction decides which sensor ends the crossing and
	// which way a recovery must finish it. Each initialises FALSE, so neither can
	// survive a download asserting what the sensors contradict - a four-valued phase
	// did, and it put two pallets on one carriage.
	_LoadingIn			: BOOL;		// drawing a pallet aboard; ends at B_Detect
	_UnloadingOut		: BOOL;		// pushing a pallet off;    ends at B_Exit
	// Edge detectors for the clearing rules. A level cannot be used: during an
	// outbound crossing B_Detect is still made while the pallet leaves, and B_Exit
	// may still be made by the previous pallet when the next crossing commits.
	// Edges are also the only witness a stop cannot erase - an earlier version used
	// the live belt command and deadlocked, because Stopping clears it.
	DetectEdge			: R_TRIG;
	ExitEdge			: R_TRIG;
	_NextCanAccept		: BOOL;		// the successor can physically accept a pallet
	_PayloadIncoming	: BOOL;		// the predecessor is releasing a pallet to us

	// --- Diagnostics --------------------------------------------------------
	// 0 none  1 no home  2 pallet never arrived aboard  3 travel failed
	// 4 pallet never left
	// Raised while finishing an interrupted crossing in Resetting:
	// 5 reset: pallet never came aboard   6 reset: pallet never left
	_FaultCode		: DINT;

	// --- Parameters, set by the parent in Initialize ------------------------
	// FALSE: home is the retracted (lower) end, travel is to extended (upper).
	// TRUE:  the mirror image, for the lift that returns pallets downwards.
	_ReverseDirection	: BOOL;

	_HomeTime		: TIME := T#5S;
	_LoadTime		: TIME := T#20S;	// belt running, waiting for the pallet aboard
	_TravelTime		: TIME := T#10S;
	_SettleTime		: TIME := T#500MS;	// let the pallet settle before travelling
	_UnloadTime		: TIME := T#20S;
	// How long a reset lets the line settle once this unit is home. The group runs
	// the main conveyors throughout, so loose pallets travel up against the blocking
	// stoppers and accumulate where a detect sensor can see them. Waiting a fixed
	// time cannot deadlock, which is the whole reason a reset is paced this way
	// rather than waiting on an event that may never arrive.
	_AccumulateTime	: TIME := T#5S;

	// --- HMI ----------------------------------------------------------------
	// One struct for the whole tile, extending the SPT module interface. The
	// inherited half is bridged to the base's own PackMLBaseModule_HMI in two
	// places: HMICommunication pushes Command in before the base acts on it,
	// PublishHMI copies Config and Status back out after. The Station half is this
	// block's own and is filled by PublishHMI alone.
	{ attribute 'TcHmiSymbol.AddSymbol' }
	HMI	: ST_TransferLift_HMI;
END_VAR

METHOD PROTECTED Aborting
VAR_INPUT
END_VAR
CASE SequenceState OF
	0:
		NoStateTasksToComplete	:= FALSE;
		// Stop the belt immediately. The carriage is left where it is - moving a
		// level with a pallet half on board is worse than standing still.
		//
		// Nothing is cleared. The interface is derived, and _Transferring stays
		// TRUE precisely because stopping the belt here is what leaves a pallet on
		// the boundary: Resetting needs to know that, and only the sensor that
		// completes the crossing may clear it.
		M_Conveyor.RunForward  := FALSE;
		M_Conveyor.RunBackward := FALSE;
		SequenceState		:= SequenceState + 10;

	10:
		StateTasksComplete := TRUE;
END_CASE

SUPER^.Aborting();
END_METHOD

// The carriage has reached the level it delivers to. Resolves the direction so
// the step chain reads identically for both instances.
PROPERTY PRIVATE AtFar : BOOL
GET
IF _ReverseDirection THEN
	AtFar := Y_Lift.Retracted;
ELSE
	AtFar := Y_Lift.Extended;
END_IF
END_GET
END_PROPERTY

// The carriage has reached the level it loads from.
PROPERTY PRIVATE AtHome : BOOL
GET
IF _ReverseDirection THEN
	AtHome := Y_Lift.Extended;
ELSE
	AtHome := Y_Lift.Retracted;
END_IF
END_GET
END_PROPERTY

// This lift can physically take a pallet right now. The predecessor gates its
// release on this, and it is the whole of the readiness contract.
//
// DERIVED, NOT ASSIGNED - and that is what fixed the collision. The old _Ready was
// written only inside the Execute step chain, so a reset that homed the carriage
// with a pallet still aboard came back announcing an empty lift and the stopper
// released a second pallet into it. Computed from the carriage position, the
// detect sensor and the transfer latch, this is correct in every PackML state and
// every mode, which is also why the reset recovery can use the same contract.
PROPERTY CanAccept : BOOL
GET
CanAccept := AtHome
	AND NOT B_Detect.Active
	AND NOT Transferring
	AND (_FaultCode = 0);
END_GET
END_PROPERTY

METHOD PROTECTED Clearing
VAR_INPUT
END_VAR
CASE SequenceState OF
	0:
		NoStateTasksToComplete := FALSE;
		_FaultCode := 0;
		SequenceState := SequenceState + 10;

	10:
		IF Y_Lift.Reset()
			AND B_Detect.Reset()
			AND B_Exit.Reset()
			AND M_Conveyor.Reset() THEN
			SequenceState := SequenceState + 10;
		END_IF

	20:
		StateTasksComplete := TRUE;
END_CASE

SUPER^.Clearing();
END_METHOD

METHOD PUBLIC CyclicLogic
VAR_INPUT
END_VAR
IF NOT _InitComplete THEN
	_InitComplete := Initialize();
	RETURN;
END_IF

// Nothing to copy: every output is linked to its terminal at the instance
// declaration in FG_Transport.

// THE TRANSFER LATCHES ARE RESOLVED BY SENSOR EDGES, IN EVERY STATE. B_Detect ends
// an inbound crossing, B_Exit an outbound one; each latch carries its direction.
// EDGES, NOT LEVELS, AND NOT THE BELT COMMAND. Using the live belt direction as
// the witness deadlocked the machine: Stopping and Aborting clear the belt command
// immediately, destroying the witness, and the latch could never clear.
DetectEdge(CLK := B_Detect.Active);
ExitEdge(CLK := B_Exit.Active);

IF _LoadingIn AND DetectEdge.Q THEN
	_LoadingIn := FALSE;
END_IF
IF _UnloadingOut AND ExitEdge.Q THEN
	_UnloadingOut := FALSE;
END_IF

// TWO STATES MAY DRIVE THE CARRIAGE BELT: Execute, and Resetting - which finishes
// an interrupted transfer. In every other state a run request is stale.
// THIS GUARD RUNS BEFORE SUPER^.CyclicLogic(), so it does not merely veto the
// output for a scan - it WIPES the request Resetting set on the previous scan.
// Leaving a state out of this condition makes its belt commands invisible to the
// drive: it looks exactly like a conveyor commanded and never moving.
IF (_CurrentState <> E_PMLState.ePMLState_Execute)
	AND (_CurrentState <> E_PMLState.ePMLState_Resetting) THEN
	M_Conveyor.RunForward := FALSE;
	M_Conveyor.RunBackward := FALSE;
END_IF

// THE CARRIAGE BELT MAY ONLY RUN WHILE THE CARRIAGE IS AT A LEVEL. Between levels
// it drives the pallet into a fixed edge. A physical property, so it is enforced
// here for every state and mode - including Manual, where the operator jogs.
// It is also what the transfer latches rest on: a crossing can only START at a
// level, so a set latch is proof the carriage is in position.
IF NOT (AtHome OR AtFar) THEN
	M_Conveyor.RunForward := FALSE;
	M_Conveyor.RunBackward := FALSE;
END_IF

SUPER^.CyclicLogic();

// After the base, so the published struct carries this scan's state and
// this scan's HMI permission rather than last scan's.
PublishHMI();
END_METHOD

METHOD PROTECTED Execute
VAR_INPUT
END_VAR
VAR_INST
	HomeTimer		: TON;
	LoadTimer		: TON;
	SettleTimer		: TON;
	TravelTimer		: TON;
	UnloadTimer		: TON;
END_VAR
// The ring runs continuously, so this state loops instead of completing.
//
// AtHome / AtFar resolve the direction once, so the step chain below reads the
// same for both instances and only Initialize differs between them.

CASE _CurrentMode OF

	//============================= PRODUCTION =================================
	E_PMLUnitMode.ePMLUnitMode_Production:

		CASE SequenceState OF
			0:	// Return to the loading level with the belt stopped - but only if
				// the carriage is actually clear. Commanding a level change under
				// a pallet is the one thing this unit must never do blindly, and
				// this step is where that command is issued.
				//
				// The sensor decides. There is no remembered occupancy to consult
				// and nothing to publish: CanAccept is derived and is already
				// correct before this step runs.
				NoStateTasksToComplete	:= FALSE;
				M_Conveyor.RunForward  := FALSE;
				M_Conveyor.RunBackward := FALSE;

				IF B_Detect.Active THEN
					// A pallet is aboard. Do not command the carriage anywhere:
					// resume the delivery from the settle step, which is where the
					// normal load path hands over once a pallet is on board.
					SequenceState	:= 40;
				ELSE
					IF _ReverseDirection THEN
						Y_Lift.Extend();
					ELSE
						Y_Lift.Retract();
					END_IF
					SequenceState := SequenceState + 10;
				END_IF

			10:
				IF AtHome THEN
					SequenceState	:= SequenceState + 10;
				ELSIF HomeTimer.Q THEN
					_FaultCode := 1;
					ChangeState(E_PMLCommand.ePMLCommand_Hold);
				END_IF

			20:	// Wait to be told a pallet is coming. Unlike every other unit a
				// lift does not self-detect here - it has to run its belt to
				// draw the pallet aboard, so it must be told first.
				// B_Detect IS TESTED FIRST, and that ordering is load bearing. A
				// latch armed while its ending sensor is already made can never see
				// a rising edge, so it would stay TRUE for ever. Testing the sensor
				// first guarantees _LoadingIn is only ever armed with B_Detect
				// clear, which guarantees the edge that clears it.
				IF B_Detect.Active THEN
					// Already aboard - unannounced, or the announcement arrived with
					// the pallet. Nothing is crossing; go straight to settle.
					SequenceState		:= 40;
				ELSIF _PayloadIncoming THEN
					M_Conveyor.RunBackward := TRUE;
					// The inbound crossing starts here. Until B_Detect confirms, the
					// pallet spans the carriage and the fixed conveyor and nothing
					// may change level. Cleared on the B_Detect edge in CyclicLogic.
					_LoadingIn			:= TRUE;
					SequenceState		:= SequenceState + 10;
				END_IF

			30:	// Belt running, waiting for the pallet to arrive on the carriage.
				// _Transferring has already been cleared by B_Detect in CyclicLogic.
				IF B_Detect.Active THEN
					M_Conveyor.RunBackward := FALSE;
					SequenceState		:= SequenceState + 10;
				ELSIF LoadTimer.Q THEN
					M_Conveyor.RunBackward := FALSE;
					_FaultCode			:= 2;
					ChangeState(E_PMLCommand.ePMLCommand_Hold);
				END_IF

			40:	// Let the pallet settle before the carriage moves
				IF SettleTimer.Q THEN
					SequenceState := SequenceState + 10;
				END_IF

			50:	// Travel to the far level
				IF _ReverseDirection THEN
					Y_Lift.Retract();
				ELSE
					Y_Lift.Extend();
				END_IF
				IF AtFar THEN
					SequenceState := SequenceState + 10;
				ELSIF TravelTimer.Q THEN
					_FaultCode := 3;
					ChangeState(E_PMLCommand.ePMLCommand_Hold);
				END_IF

			60:	// The successor must be able to accept before anything is pushed
				// at it
				IF _NextCanAccept THEN
// Commit HERE, once, on the transition. Setting it inside step 70
					// would re-assert it on the scan CyclicLogic clears it, latching
					// it TRUE for ever. Armed only if B_Exit is clear: a latch armed
					// under an already-made sensor never sees its clearing edge.
					_UnloadingOut	:= NOT B_Exit.Active;
					SequenceState	:= SequenceState + 10;
				END_IF

			70:	// Push the pallet off. No announcement to the successor - it
				// picks the pallet up on its own detect sensor. _Transferring is
				// cleared by B_Exit in CyclicLogic.
				M_Conveyor.RunForward  := TRUE;
				IF B_Exit.Active THEN
					SequenceState := SequenceState + 10;
				ELSIF UnloadTimer.Q THEN
					M_Conveyor.RunForward  := FALSE;
					_FaultCode			:= 4;
					ChangeState(E_PMLCommand.ePMLCommand_Hold);
				END_IF

			80:	// Stop the belt before returning home.
				// DELIBERATE DIFFERENCE FROM SIL: SequenceTransferLift leaves the
				// belt running through the return travel and only clears it when
				// Idle re-runs. Carrying a driven belt through a level change can
				// drag whatever is on it, and nothing in the context asks for it.
				M_Conveyor.RunForward  := FALSE;
				SequenceState		:= 0;
		END_CASE

	//======================= MAINTENANCE & MANUAL =============================
	E_PMLUnitMode.ePMLUnitMode_Maintenance, E_PMLUnitMode.ePMLUnitMode_Manual:
		// Nothing to drive. Both devices honour their own HMI structs, and both belt
		// directions are offered by hand. Nothing is assigned: the interface is derived
		// from the sensors, so it keeps telling the truth while an operator works. A
		// crossing created by jogging is invisible to this unit - Manual is supervised.
		;
END_CASE

SUPER^.Execute();

HomeTimer(	IN := (SequenceState = 10),							PT := _HomeTime);
LoadTimer(	IN := (SequenceState = 30),							PT := _LoadTime);
SettleTimer(IN := (SequenceState = 40),							PT := _SettleTime);
TravelTimer(IN := (SequenceState = 50),							PT := _TravelTime);
UnloadTimer(IN := (SequenceState = 70),							PT := _UnloadTime);
END_METHOD

// 0 none  1 no home  2 pallet never arrived aboard  3 travel failed
// 4 pallet never left
// Raised by the recovery in Resetting:
// 5 reset: pallet never finished loading      6 reset: pallet never left
// 7 reset: travel to the delivery level failed
// 8 reset: successor still occupied - the pallet cannot be handed over
PROPERTY FaultCode : DINT
GET
FaultCode := _FaultCode;
END_GET
END_PROPERTY

METHOD PROTECTED HMICommunication
VAR_INPUT
END_VAR
// The command half of the HMI bridge; PublishHMI is the status half.
// The base calls this immediately before ModeControl() and StateControl(), which
// is the only point at which an operator command can still reach this scan's
// state machine. See FB_TransferIndex.HMICommunication for the full reasoning.
PackMLBaseModule_HMI.Command := HMI.Command;

SUPER^.HMICommunication();

// The base clears a latch by writing back the value it acted on.
HMI.Command := PackMLBaseModule_HMI.Command;
END_METHOD

METHOD PROTECTED Initialize : BOOL;
VAR
END_VAR
Initialize := FALSE;

CASE DescendantSequenceState OF
	0:
		RegisterComponent(B_Detect);
		RegisterComponent(B_Exit);
		RegisterComponent(Y_Lift);

		// The carriage belt is a component owned directly by this lift.
		RegisterComponent(M_Conveyor);

		_LogModeChanges		:= FALSE;
		_LogStateChanges	:= FALSE;
		DescendantSequenceState := DescendantSequenceState + 10;

	10:
		// A level change is a long stroke - these are travel alarms, not pacing.
		Y_Lift.ExtendTime	:= 10000.0;
		Y_Lift.RetractTime	:= 10000.0;
		DescendantSequenceState := DescendantSequenceState + 10;

	20:
		IF SUPER^.Initialize() THEN
			DescendantSequenceState := DescendantSequenceState + 10;
		END_IF

	30:
		Initialize := TRUE;
END_CASE
END_METHOD

// The successor's CanAccept, wired in by the parent.
//
// One channel, used by both Execute and the recovery in Resetting. The separate
// NextOccupied input that the recovery needed before is gone: CanAccept is derived
// and therefore answers in every state, so there is nothing left for a second
// channel to say.
PROPERTY NextCanAccept : BOOL
SET
_NextCanAccept := NextCanAccept;
END_SET
END_PROPERTY

// This lift is physically carrying or handling a pallet.
//
// Derived, like CanAccept: the detect sensor, or a crossing that has been started
// and not yet confirmed finished. The latch half is not redundant - a pallet drawn
// half onto the carriage has not reached B_Detect, and that is precisely the state
// in which nobody may send another one and the carriage may not change level.
//
// There is no remembered occupancy behind this, so there is nothing for a state
// change or a program download to falsify.
PROPERTY Occupied : BOOL
GET
Occupied := B_Detect.Active OR Transferring;
END_GET
END_PROPERTY

// The predecessor is releasing a pallet to us. On a lift this is not a courtesy
// notice - it is the command that starts the belt drawing the pallet aboard.
PROPERTY PayloadIncoming : BOOL
SET
_PayloadIncoming := PayloadIncoming;
END_SET
END_PROPERTY

ACTION PublishHMI:
// Everything an operator tile needs from this unit, in one struct.
//
// Called from CyclicLogic AFTER SUPER^.CyclicLogic(), so _CurrentState and the
// base's HMIControlAvailable are this scan's values and not last scan's.
//
// The carriage belt publishes itself - M_Conveyor is an FB_AbstractBinaryDrive and
// has its own HMI struct, which the tile binds to as a second parameter.

// --- Inherited half ---------------------------------------------------------
// Straight copies of the struct the SPT base maintains - Config carries Name and
// the logging toggles, Status carries Busy, Error, ErrorID, Mode, State and
// HMIControlAvailable. The last is the gate for the jog buttons on the tile,
// granted in ePMLUnitMode_Manual only.
HMI.Config		:= PackMLBaseModule_HMI.Config;
HMI.Status		:= PackMLBaseModule_HMI.Status;

HMI.StateName			:= F_PMLStateName(_CurrentState);
HMI.Sequence.StepIndex	:= SequenceState;

// --- Ring handshake ---------------------------------------------------------
// A lift is a pulling station: no SendToNext, and PayloadIncoming is how the
// predecessor announces a pallet.
// The derived properties, not backing variables - the tile shows what the machine
// physically is, which is the same thing the neighbouring stations act on. The
// struct field names are unchanged so the existing panel bindings still resolve.
HMI.Station.Ready					:= CanAccept;
HMI.Station.Occupied				:= Occupied;
HMI.Station.NextReady				:= _NextCanAccept;
HMI.Station.PayloadIncoming		:= _PayloadIncoming;
HMI.Station.ReverseDirection		:= _ReverseDirection;

// --- Diagnostics ------------------------------------------------------------
HMI.Station.FaultCode				:= _FaultCode;
END_ACTION

METHOD PROTECTED Resetting
VAR_INPUT
END_VAR
VAR_INST
	ResetCrossTimer		: TON;
	ResetHomeTimer		: TON;
	AccumulateTimer		: TON;
END_VAR
// A RESET RE-ESTABLISHES WHERE THE PALLETS ARE. IT DOES NOT DELIVER ANYTHING.
// The group runs the main conveyors throughout a reset, so loose pallets accumulate
// against the blocking stoppers. This unit only has to reach a known safe position.
//
// DELIVERING HERE DEADLOCKED. It waited for the successor's CanAccept, but a
// stopper never releases during a reset, so it could never become free. A reset
// must not depend on another unit doing what the reset forbids it to do.
//
// TWO RULES DECIDE WHAT IS SAFE HERE:
//   1. the belt may only run AT a level - enforced in CyclicLogic, not here;
//   2. a crossing can only START at a level, so a set latch is proof the carriage
//      is in position, and with no latch set nothing spans the gap.
// Hence: latch set -> finish the crossing, leave the axis alone.
//        no latch  -> move to the home level.

CASE SequenceState OF
	0:	// Route on the latches. They carry the direction, and by rule 2 a set latch
		// also means the carriage is already at a level.
		NoStateTasksToComplete	:= FALSE;

		IF Transferring THEN
			SequenceState := 10;
		ELSE
			SequenceState := 30;
		END_IF

	10:	// Finish the crossing in the direction it was already going. Waits on the
		// SENSOR, not on the latch: the latch serves the interface and is cleared by
		// the same edge, and keeping the chain independent of it means a latch that
		// somehow failed to clear cannot strand the sequence as well.
		
		ResetCrossTimer(IN := TRUE, PT := SEL(_LoadingIn, _UnloadTime, _LoadTime));
		
		IF _LoadingIn THEN
			M_Conveyor.RunBackward := TRUE;
			IF B_Detect.Active THEN
				M_Conveyor.RunBackward := FALSE;
				SequenceState := 20;
			ELSIF ResetCrossTimer.Q THEN
				M_Conveyor.RunBackward := FALSE;
				_FaultCode := 5;
				ChangeState(E_PMLCommand.ePMLCommand_Hold);
			END_IF
		ELSE
			M_Conveyor.RunForward := TRUE;
			IF B_Exit.Active THEN
				M_Conveyor.RunForward := FALSE;
				SequenceState := 20;
			ELSIF ResetCrossTimer.Q THEN
				M_Conveyor.RunForward := FALSE;
				_FaultCode := 6;
				ChangeState(E_PMLCommand.ePMLCommand_Hold);
			END_IF
		END_IF	
		

	20:	// The crossing is over, however it ended. Clearing both latches here is the
		// reset doing its job: it re-establishes the state rather than inheriting a
		// latch whose sensor edge was missed while the machine was stopped.
		ResetCrossTimer(IN := FALSE, PT := SEL(_LoadingIn, _UnloadTime, _LoadTime));
		_LoadingIn		:= FALSE;
		_UnloadingOut	:= FALSE;
		SequenceState	:= 30;

	30:	// Nothing spans the gap now, so the axis may move. Belt off first.
		M_Conveyor.RunForward  := FALSE;
		M_Conveyor.RunBackward := FALSE;
		IF _ReverseDirection THEN
			Y_Lift.Extend();
		ELSE
			Y_Lift.Retract();
		END_IF
		SequenceState := 40;

	40:
		IF AtHome THEN
			SequenceState := 50;
		ELSIF ResetHomeTimer.Q THEN
			_FaultCode := 1;
			ChangeState(E_PMLCommand.ePMLCommand_Hold);
		END_IF

	50:	// Let the line settle before declaring the reset done, so production starts
		// from an accumulated, sensed state rather than a moving one. A fixed wait
		// cannot deadlock; waiting on an event that may never arrive can, which is
		// what went wrong before.
		IF AccumulateTimer.Q THEN
			SequenceState := 60;
		END_IF

	60:
		StateTasksComplete := TRUE;
END_CASE

SUPER^.Resetting();

// SEL(G, IN0, IN1) yields IN0 when G is FALSE - so an inbound crossing is bounded
// by the load time and an outbound one by the unload time.

ResetHomeTimer(	IN := (SequenceState = 40),		PT := _HomeTime);
AccumulateTimer(IN := (SequenceState = 50),		PT := _AccumulateTime);
END_METHOD

// FALSE: loads at the retracted (lower) end and delivers to the extended end.
// TRUE: the mirror image. Set once by the parent in Initialize.
PROPERTY ReverseDirection : BOOL
SET
_ReverseDirection := ReverseDirection;
END_SET
END_PROPERTY

METHOD PROTECTED Stopping
VAR_INPUT
END_VAR
CASE SequenceState OF
	0:
		NoStateTasksToComplete	:= FALSE;
		// Nothing to clear - see Aborting.
		M_Conveyor.RunForward  := FALSE;
		M_Conveyor.RunBackward := FALSE;
		SequenceState		:= SequenceState + 10;

	10:
		StateTasksComplete := TRUE;
END_CASE

SUPER^.Stopping();
END_METHOD

// A payload is crossing the carriage boundary in either direction, so the carriage
// must not change level. The two directional latches read as one fact wherever the
// direction does not matter.
PROPERTY PRIVATE Transferring : BOOL
GET
Transferring := _LoadingIn OR _UnloadingOut;
END_GET
END_PROPERTY

END_FUNCTION_BLOCK

// ---- Library/POUs/FB_AbstractBinaryDrive.TcPOU
// Reusable two-direction conveyor drive SPT component.
FUNCTION_BLOCK FB_AbstractBinaryDrive EXTENDS FB_ComponentBase
VAR
	_Forward AT %Q* : BOOL;
	_Backward AT %Q* : BOOL;
	_DriveActive AT %I* : BOOL;
	_RunForward : BOOL;
	_RunBackward : BOOL;
	_FaultCode : UDINT;
	_StartTime : TIME := T#2S;
	StartTimer : TON;
	{ attribute 'TcHmiSymbol.AddSymbol' }
	HMI : ST_AbstractBinaryDrive_HMI;
END_VAR

PROPERTY Active : BOOL
GET
Active := _DriveActive;
END_GET
END_PROPERTY

METHOD PUBLIC CyclicLogic
VAR_INPUT END_VAR
IF NOT _InitComplete THEN
	_InitComplete := Initialize();
	RETURN;
END_IF

_Forward := _RunForward AND NOT _RunBackward AND (_FaultCode = 0);
_Backward := _RunBackward AND NOT _RunForward AND (_FaultCode = 0);
StartTimer(IN := (_Forward OR _Backward) AND NOT _DriveActive, PT := _StartTime);
IF StartTimer.Q THEN
	_FaultCode := 1;
	_Forward := FALSE;
	_Backward := FALSE;
END_IF

_Busy := (_Forward OR _Backward) AND NOT _DriveActive;
_Error := _FaultCode <> 0;
_ErrorID := _FaultCode;
SUPER^.CyclicLogic();

// Device config and status only. The inherited Config / Command / Status half of
// HMI is a mirror of ComponentBase_HMI and is bridged in HMICommunication.
HMI.DeviceConfig.StartTime := _StartTime;
HMI.Device.Running := _Forward OR _Backward;
HMI.Device.Active := _DriveActive;
HMI.Device.Forward := _Forward;
HMI.Device.Backward := _Backward;
HMI.Device.Error := _Error;
HMI.Device.ErrorCode := _FaultCode;
END_METHOD

PROPERTY FaultCode : UDINT
GET
FaultCode := _FaultCode;
END_GET
END_PROPERTY

METHOD PROTECTED HMICommunication
VAR_INPUT END_VAR
// HMI is a published mirror of the base's own ComponentBase_HMI - carry operator
// intent in before the base looks, and its answers back out afterwards.
ComponentBase_HMI.Command := HMI.Command;

SUPER^.HMICommunication();

HMI.Config	:= ComponentBase_HMI.Config;
HMI.Status	:= ComponentBase_HMI.Status;
HMI.Command	:= ComponentBase_HMI.Command;

IF HMI.DeviceConfig.StartTime > T#0S THEN
	_StartTime := HMI.DeviceConfig.StartTime;
END_IF
IF ComponentBase_HMI.Status.HMIControlAvailable THEN
	_RunForward := HMI.DeviceCommand.RunForward;
	_RunBackward := HMI.DeviceCommand.RunBackward;
ELSE
	HMI.DeviceCommand.RunForward := _RunForward;
	HMI.DeviceCommand.RunBackward := _RunBackward;
END_IF
END_METHOD

METHOD PROTECTED Initialize : BOOL
VAR_INPUT END_VAR
Initialize := SUPER^.Initialize();
END_METHOD

METHOD PUBLIC Reset : BOOL
VAR_INPUT END_VAR
Reset := SUPER^.Reset();
IF Reset THEN
	_FaultCode := 0;
	_RunForward := FALSE;
	_RunBackward := FALSE;
	_Forward := FALSE;
	_Backward := FALSE;
END_IF
END_METHOD

PROPERTY RunBackward : BOOL
GET
RunBackward := _RunBackward;
END_GET
SET
_RunBackward := RunBackward;
END_SET
END_PROPERTY

PROPERTY RunForward : BOOL
GET
RunForward := _RunForward;
END_GET
SET
_RunForward := RunForward;
END_SET
END_PROPERTY

PROPERTY StartTime : TIME
GET
StartTime := _StartTime;
END_GET
SET
_StartTime := StartTime;
END_SET
END_PROPERTY

END_FUNCTION_BLOCK

// ---- Modules/11 FG_01/FG_01.TcPOU
// FG_01 - identify, mark, verify identity. Nine SPT components.
// Triggered by Index01; reports OperationDone. A wrong serial aborts (fault 1).
// Y_Gate1/Y_Gate2 CLOSE on Extend - the opposite sense to a transport stopper.
// Twin side: FB_Camera in OC_SIM - both halves must agree on the bit layout.
// Contract: _workflow/reference/fg-01-behaviour.md
FUNCTION_BLOCK FG_01 EXTENDS FB_PackML_BaseModule
VAR
	{ attribute 'TcHmiSymbol.AddSymbol' }
	Y_Gripper		: FB_DoubleSolenoidFeedback := (Name := 'Y_Gripper');
	{ attribute 'TcHmiSymbol.AddSymbol' }
	Y_Platform		: FB_DoubleSolenoidFeedback := (Name := 'Y_Platform');
	{ attribute 'TcHmiSymbol.AddSymbol' }
	Y_ReaderWindow	: FB_DoubleSolenoidFeedback := (Name := 'Y_ReaderWindow');
	P_Camera		: FB_AbstractCamera := (Name := 'P_Camera');
	Y_LaserMark		: FB_AbstractLightSource := (Name := 'Y_LaserMark');
	{ attribute 'TcHmiSymbol.AddSymbol' }
	Y_Gate1			: FB_SingleSolenoidFeedback := (Name := 'Y_Gate1');
	{ attribute 'TcHmiSymbol.AddSymbol' }
	Y_Gate2			: FB_SingleSolenoidFeedback := (Name := 'Y_Gate2');
	{ attribute 'TcHmiSymbol.AddSymbol' }
	B_SafetyGate1	: FB_DigitalSensor := (Name := 'B_SafetyGate1');
	{ attribute 'TcHmiSymbol.AddSymbol' }
	B_SafetyGate2	: FB_DigitalSensor := (Name := 'B_SafetyGate2');

	// Group level fault - see ST_FG_01_Identify_Status. Cleared in Clearing.
	_FaultCode		: DINT;
	// The verdict of the last completed read, latched so the panel still shows it
	// once ResultValid has dropped.
	_LastResultOK	: BOOL;

	{ attribute 'TcHmiSymbol.AddSymbol' }
	HMI : ST_HMI_FG_01;
END_VAR

METHOD PROTECTED Aborting
VAR_INPUT
END_VAR
CASE SequenceState OF
	0:
		NoStateTasksToComplete	:= FALSE;
		// Laser first - it is the only hazardous output here.

		Y_LaserMark.Disable();
		P_Camera.Disable();
		SequenceState			:= SequenceState + 10;

	10:	// Shield the optics. The gripper keeps its grip on purpose - releasing a
		// clamped payload on abort would drop it.
		Y_ReaderWindow.Retract();
		IF Y_ReaderWindow.Retracted THEN
			SequenceState := SequenceState + 10;
		END_IF

	20:
		StateTasksComplete := TRUE;
END_CASE

SUPER^.Aborting();
END_METHOD

METHOD PROTECTED Clearing
VAR_INPUT
END_VAR
CASE SequenceState OF
	0:
		NoStateTasksToComplete := FALSE;
		// Cleared by the act of clearing, not by the condition going away.
		_FaultCode := 0;
		SequenceState := SequenceState + 10;

	10:	// Clear latched component alarms - the solenoid travel timeouts latch.
		IF Y_Gripper.Reset()
			AND Y_Platform.Reset()
			AND Y_ReaderWindow.Reset()
			AND P_Camera.Reset()
			AND Y_LaserMark.Reset()
			AND Y_Gate1.Reset()
			AND Y_Gate2.Reset()
			AND B_SafetyGate1.Reset()
			AND B_SafetyGate2.Reset() THEN
			SequenceState := SequenceState + 10;
		END_IF

	20:
		StateTasksComplete := TRUE;
END_CASE

SUPER^.Clearing();
END_METHOD

METHOD PUBLIC CyclicLogic
VAR_INPUT
END_VAR
IF NOT _InitComplete THEN
	_InitComplete := Initialize();
	RETURN;
END_IF

// No process image copy step: component members map straight to terminal channels.
SUPER^.CyclicLogic();

PublishStatus();
END_METHOD

METHOD PROTECTED Execute
VAR_INPUT
END_VAR
VAR_INST
	ClampSettleTimer	: TON;
	MarkTimer			: TON;
	ReadyTimer			: TON;
	ShotTimer			: TON;
END_VAR
// Y_Platform is deliberately absent: it positions the laser head in service
// only and is never actuated during the cycle.
CASE _CurrentMode OF

	//============================= PRODUCTION =================================
	E_PMLUnitMode.ePMLUnitMode_Production:

		CASE SequenceState OF
			0:
				NoStateTasksToComplete	:= FALSE;
				Y_LaserMark.Disable();
				// Camera on at the start, not at the read: it has the whole
				// gate-clamp-mark sequence to come Ready in.
				P_Camera.Enable();
				P_Camera.ClearTrigger();
				SequenceState			:= SequenceState + 10;

			10:	// Shut the cell. Both gates commanded on one scan, both limits
				// waited on, so they travel together.
				Y_Gate1.Extend();
				Y_Gate2.Extend();
				IF Y_Gate1.Extended AND Y_Gate2.Extended AND B_SafetyGate1.Active AND B_SafetyGate2.Active THEN
					SequenceState := SequenceState + 10;
				END_IF

			20:	// Clamp the payload
				Y_Gripper.Extend();
				SequenceState := SequenceState + 10;

			30:	// Let the clamp settle before firing
				IF ClampSettleTimer.Q THEN
					SequenceState := SequenceState + 10;
				END_IF

			40:	// Mark. The gates were proven at step 10 and nothing opens them until
				// step 120, so there is no per-scan permissive here by design.
				Y_LaserMark.Enable();
				IF MarkTimer.Q THEN
					Y_LaserMark.Disable();
					SequenceState	:= SequenceState + 10;
				END_IF

			50:	// Open the window for the read
				Y_ReaderWindow.Extend();
				SequenceState := SequenceState + 10;

			60:	// Window open. Wait for Ready; a timeout here is a wiring or
				// device fault, not a slow start.
				IF Y_ReaderWindow.Extended THEN
					IF P_Camera.Ready THEN
						SequenceState := SequenceState + 10;
					ELSIF ReadyTimer.Q THEN
						_FaultCode := 2;
						AbortImmediate();
					END_IF
				END_IF

			70:	// Trigger. ResultValid also acknowledges: a fast camera can raise
				// and drop Busy inside one scan.
				P_Camera.Trigger();
				IF P_Camera.DeviceBusy OR P_Camera.ResultValid THEN
					SequenceState := SequenceState + 10;
				ELSIF ShotTimer.Q THEN
					_FaultCode := 3;
					AbortImmediate();
				END_IF

			80:	// Read the verdict. It stands until the trigger is released.
				IF P_Camera.ResultValid THEN
					_LastResultOK := P_Camera.ResultOK;
					IF P_Camera.ResultOK THEN
						SequenceState := SequenceState + 10;
					ELSE
						_FaultCode := 1;
						AbortImmediate();
					END_IF
				ELSIF ShotTimer.Q THEN
					_FaultCode := 3;
					AbortImmediate();
				END_IF

			90:	// Release the trigger - that is what tells the camera its verdict
				// was read. Enable stays on to the end of the cycle.
				P_Camera.ClearTrigger();
				SequenceState := SequenceState + 10;

			100: // Shield the optics again
				Y_ReaderWindow.Retract();
				IF Y_ReaderWindow.Retracted THEN
					SequenceState := SequenceState + 10;
				END_IF

			110: // Release the payload
				Y_Gripper.Retract();
				IF Y_Gripper.Retracted THEN
					SequenceState := SequenceState + 10;
				END_IF

			120: // Open the cell, both gates together. Only now: opening while the
				// payload is clamped would expose a held part.
				Y_Gate1.Retract();
				Y_Gate2.Retract();
				IF Y_Gate1.Retracted AND Y_Gate2.Retracted AND NOT B_SafetyGate1.Active AND NOT B_SafetyGate2.Active THEN
					SequenceState := SequenceState + 10;
				END_IF

			130: // Execute is the one acting state that does not self-complete.
				// StateComplete() would be wrong here.
				P_Camera.Disable();
				ChangeState(E_PMLCommand.ePMLCommand_Complete);
		END_CASE

	//======================= MAINTENANCE & MANUAL =============================
	E_PMLUnitMode.ePMLUnitMode_Maintenance, E_PMLUnitMode.ePMLUnitMode_Manual:
		// No group sequence. Y_Platform and P_Camera stay reachable
			// through their own component HMI control.
		;
END_CASE

SUPER^.Execute();

// These conditions name step numbers: renumbering a step moves its timer too.
ClampSettleTimer(IN := (SequenceState = 30) AND Y_Gripper.Extended,	PT := T#500MS);
MarkTimer(IN := SequenceState = 40,									PT := T#1S);

// ReadyTimer is armed on the WINDOW BEING OPEN, not on the step alone. Step 50
// extends and advances on the same scan, so arming on the step would let a slow
// window burn the camera's budget and raise fault 2 for a pneumatic fault.
ReadyTimer(IN := (SequenceState = 60) AND Y_ReaderWindow.Extended,	PT := T#2S);
ShotTimer(IN := (SequenceState = 70) OR (SequenceState = 80),		PT := T#3S);
END_METHOD

METHOD PROTECTED HMICommunication
VAR_INPUT
END_VAR
// Command half of the HMI bridge; PublishStatus is the status half. MUST be in
// this method: the base calls it immediately before ModeControl() and
// StateControl(), and reads its own PackMLBaseModule_HMI.Command, never ours.
PackMLBaseModule_HMI.Command := HMI.Command;

SUPER^.HMICommunication();

// The base clears a latch by writing back the value it acted on.
HMI.Command := PackMLBaseModule_HMI.Command;
END_METHOD

METHOD PROTECTED Initialize : BOOL;
VAR
END_VAR
Initialize := FALSE;

CASE DescendantSequenceState OF
	0:
		RegisterComponent(Y_Gripper);
		RegisterComponent(Y_Platform);
		RegisterComponent(Y_ReaderWindow);
		RegisterComponent(P_Camera);
		RegisterComponent(Y_LaserMark);
		RegisterComponent(Y_Gate1);
		RegisterComponent(Y_Gate2);
		RegisterComponent(B_SafetyGate1);
		RegisterComponent(B_SafetyGate2);

		_LogModeChanges		:= FALSE;
		_LogStateChanges	:= TRUE;
		HMI.Config.Name		:= THIS^._Name;
		DescendantSequenceState := DescendantSequenceState + 10;

	10:
		// Travel timeouts in ms. They alarm on a jam; they do not pace the cycle.
		Y_Gripper.ExtendTime		:= 2000.0;
		Y_Gripper.RetractTime		:= 2000.0;
		Y_Platform.ExtendTime		:= 3000.0;
		Y_Platform.RetractTime		:= 3000.0;
		Y_ReaderWindow.ExtendTime	:= 2000.0;
		Y_ReaderWindow.RetractTime	:= 2000.0;
		// The gates are a longer stroke than the small pneumatics above.
		Y_Gate1.ExtendTime			:= 3000.0;
		Y_Gate1.RetractTime			:= 3000.0;
		Y_Gate2.ExtendTime			:= 3000.0;
		Y_Gate2.RetractTime			:= 3000.0;
		DescendantSequenceState := DescendantSequenceState + 10;

	20:
		IF SUPER^.Initialize() THEN
			DescendantSequenceState := DescendantSequenceState + 10;
		END_IF

	30:
		Initialize := TRUE;
END_CASE
END_METHOD

ACTION PublishStatus:
// Status half of the HMI bridge. Called AFTER SUPER^.CyclicLogic(), so every
// field is this scan's. Copy the base struct wholesale - setting fields one by
// one leaves Busy, Error, ErrorID and HMIControlAvailable at zero.
// The nine devices publish themselves; what is added here is what none owns.
HMI.Config		:= PackMLBaseModule_HMI.Config;
HMI.Status		:= PackMLBaseModule_HMI.Status;

HMI.StateName				:= F_PMLStateName(_CurrentState);
HMI.Sequence.StepIndex		:= SequenceState;
HMI.Identify.FaultCode		:= _FaultCode;
HMI.Identify.LastResultOK	:= _LastResultOK;
END_ACTION

METHOD PROTECTED Resetting
VAR_INPUT
END_VAR
// Home: nothing energised, optics shielded, payload released.

CASE SequenceState OF
	0:
		NoStateTasksToComplete	:= FALSE;
		Y_LaserMark.Disable();
		P_Camera.Disable();
		SequenceState			:= SequenceState + 10;

	10:	// Shield the optics first
		Y_ReaderWindow.Retract();
		IF Y_ReaderWindow.Retracted THEN
			SequenceState := SequenceState + 10;
		END_IF

	20:	// Then release
		Y_Gripper.Retract();
		IF Y_Gripper.Retracted THEN
			SequenceState := SequenceState + 10;
		END_IF

	30:	// Gates last, once the payload is free. Retracted is home, which is OPEN.
		Y_Gate1.Retract();
		Y_Gate2.Retract();
		IF Y_Gate1.Retracted AND Y_Gate2.Retracted THEN
			SequenceState := SequenceState + 10;
		END_IF

	40:
		StateTasksComplete := TRUE;
END_CASE

SUPER^.Resetting();
END_METHOD

METHOD PROTECTED Stopping
VAR_INPUT
END_VAR
// Stop leaves the payload clamped and optics shielded, so the cycle resumes
// after a reset without re-fixturing.

CASE SequenceState OF
	0:
		NoStateTasksToComplete	:= FALSE;
		Y_LaserMark.Disable();
		P_Camera.Disable();
		SequenceState			:= SequenceState + 10;

	10:
		Y_ReaderWindow.Retract();
		IF Y_ReaderWindow.Retracted THEN
			SequenceState := SequenceState + 10;
		END_IF

	20:
		StateTasksComplete := TRUE;
END_CASE

SUPER^.Stopping();
END_METHOD

END_FUNCTION_BLOCK

// ---- Library/POUs/FB_AbstractCamera.TcPOU
// ============================================================================
// Inspection camera - the CONTROL side of a vision sensor. Three instances, all
// named P_Camera: FG_01, FG_02, FG_05. One device, one bit layout; the stations
// differ only in which payload key their twin reads and what value it must be.
//
//   Output  bit 0  Enable          Input  bit 0  Ready
//           bit 1  Trigger                bit 1  Busy
//                                         bit 2  ResultValid
//                                         bit 3  ResultOK
//
// Ready is permission to trigger; ResultValid says a verdict is on the wire and
// holds it there until the trigger is released.
// The twin side is FB_Camera in OC_SIM - both halves must agree on the layout,
// and nothing checks it for you.
// READ ResultOK ONLY WHILE ResultValid. This block does not mask it for you: it
// reports both bits honestly and leaves the pairing to the caller.
FUNCTION_BLOCK FB_AbstractCamera EXTENDS FB_ComponentBase
VAR
	InputData  AT %I* : BYTE;
	OutputData AT %Q* : BYTE;
	{ attribute 'TcHmiSymbol.AddSymbol' }
	HMI : ST_AbstractCamera_HMI;
END_VAR

METHOD PUBLIC CyclicLogic
VAR_INPUT END_VAR
IF NOT _InitComplete THEN
	_InitComplete := Initialize();
	RETURN;
END_IF

// Straight off the device, not inferred. There is no error bit in this layout, so
// _Error is left alone - inventing a fault condition out of a handshake would be
// inventing the why.
_Busy := InputData.1;

SUPER^.CyclicLogic();

// Device status only. The inherited Config / Command / Status half of HMI is a
// mirror of ComponentBase_HMI and is bridged in HMICommunication.
HMI.Device.Ready		:= InputData.0;
HMI.Device.Busy			:= InputData.1;
HMI.Device.ResultValid	:= InputData.2;
HMI.Device.ResultOK		:= InputData.3;
END_METHOD

// Release the trigger, which is also what tells the camera its verdict has been
// read - ResultValid drops in response and the camera re-arms.
METHOD PUBLIC ClearTrigger
VAR_INPUT END_VAR
OutputData.1 := FALSE;
END_METHOD

// Everything off, in one call: the trigger first, so a shot is never left armed on
// a camera that is losing power on the next line.
METHOD PUBLIC Disable
VAR_INPUT END_VAR
OutputData.1 := FALSE;
OutputData.0 := FALSE;
END_METHOD

METHOD PUBLIC Enable
VAR_INPUT END_VAR
OutputData.0 := TRUE;
END_METHOD

// Ask for a shot. The camera accepts this only from Ready, so a caller that has
// not waited for Ready gets nothing rather than a queued exposure.
METHOD PUBLIC Trigger
VAR_INPUT END_VAR
OutputData.1 := TRUE;
END_METHOD

// The commanded state, read back off the control byte. The camera does not report
// "enabled" separately - Ready is its answer to having been enabled.
PROPERTY Enabled : BOOL
GET
Enabled := OutputData.0;
END_GET
END_PROPERTY

// The commanded state, read back off the control byte.
PROPERTY Triggered : BOOL
GET
Triggered := OutputData.1;
END_GET
END_PROPERTY

// Permission to trigger: the camera is enabled, idle, and holding no unread
// verdict.
PROPERTY Ready : BOOL
GET
Ready := InputData.0;
END_GET
END_PROPERTY

// The shot is in progress.
// NOT called Busy: FB_BaseFB already publishes a Busy property, and redeclaring it
// in a descendant is a compile error. Hence DeviceBusy.
PROPERTY DeviceBusy : BOOL
GET
DeviceBusy := InputData.1;
END_GET
END_PROPERTY

// A verdict is on the wire. It stands until the trigger is released, so a caller
// cannot miss it by being a scan late.
PROPERTY ResultValid : BOOL
GET
ResultValid := InputData.2;
END_GET
END_PROPERTY

// The verdict. MEANINGLESS UNLESS ResultValid IS TRUE - outside that window it
// reads FALSE because there is no result, not because the part failed.
PROPERTY ResultOK : BOOL
GET
ResultOK := InputData.3;
END_GET
END_PROPERTY

METHOD PROTECTED HMICommunication
VAR_INPUT END_VAR
// HMI is a published mirror of the base's own ComponentBase_HMI - carry operator
// intent in before the base looks, and its answers back out afterwards.
ComponentBase_HMI.Command := HMI.Command;

SUPER^.HMICommunication();

HMI.Config	:= ComponentBase_HMI.Config;
HMI.Status	:= ComponentBase_HMI.Status;
HMI.Command	:= ComponentBase_HMI.Command;

// The permissive is HMIPermissions' decision, never re-derived here or on the
// panel. With control unavailable the command struct is fed the actual output
// state, so the tile shows what the machine is doing, not what was last asked.
IF ComponentBase_HMI.Status.HMIControlAvailable THEN
	OutputData.0 := HMI.DeviceCommand.Enable;
	OutputData.1 := HMI.DeviceCommand.Trigger;
ELSE
	HMI.DeviceCommand.Enable	:= OutputData.0;
	HMI.DeviceCommand.Trigger	:= OutputData.1;
END_IF
END_METHOD

METHOD PROTECTED Initialize : BOOL
VAR_INPUT END_VAR
Initialize := SUPER^.Initialize();
END_METHOD

END_FUNCTION_BLOCK

// ---- Library/POUs/FB_AbstractLightSource.TcPOU
// Generic byte-oriented light source component.
// Output: 0 Enable. Input: 0 Enabled, 1 Error, 2..7 ErrorCode.
FUNCTION_BLOCK FB_AbstractLightSource EXTENDS FB_ComponentBase
VAR
	InputData  AT %I* : BYTE;
	OutputData AT %Q* : BYTE;
	{ attribute 'TcHmiSymbol.AddSymbol' }
	HMI : ST_AbstractLightSource_HMI;
END_VAR

METHOD PUBLIC CyclicLogic
VAR_INPUT END_VAR
IF NOT _InitComplete THEN
	_InitComplete := Initialize();
	RETURN;
END_IF

_Busy := OutputData.0 AND NOT InputData.0;
_Error := InputData.1;
_ErrorID := ErrorCode;
SUPER^.CyclicLogic();

// Device status only. The inherited Config / Command / Status half of HMI is a
// mirror of ComponentBase_HMI and is bridged in HMICommunication.
HMI.Device.Enabled := InputData.0;
HMI.Device.Error := InputData.1;
HMI.Device.ErrorCode := ErrorCode;
END_METHOD

PROPERTY DeviceError : BOOL
GET
DeviceError := InputData.1;
END_GET
END_PROPERTY

METHOD PUBLIC Disable
VAR_INPUT END_VAR
OutputData.0 := FALSE;
END_METHOD

METHOD PUBLIC Enable
VAR_INPUT END_VAR
OutputData.0 := TRUE;
END_METHOD

PROPERTY Enabled : BOOL
GET
Enabled := InputData.0;
END_GET
END_PROPERTY

PROPERTY ErrorCode : BYTE
GET
ErrorCode := SHR(InputData, 2);
END_GET
END_PROPERTY

METHOD PROTECTED HMICommunication
VAR_INPUT END_VAR
// HMI is a published mirror of the base's own ComponentBase_HMI - carry operator
// intent in before the base looks, and its answers back out afterwards.
ComponentBase_HMI.Command := HMI.Command;

SUPER^.HMICommunication();

HMI.Config	:= ComponentBase_HMI.Config;
HMI.Status	:= ComponentBase_HMI.Status;
HMI.Command	:= ComponentBase_HMI.Command;

IF ComponentBase_HMI.Status.HMIControlAvailable THEN
	OutputData.0 := HMI.DeviceCommand.Enable;
ELSE
	HMI.DeviceCommand.Enable := OutputData.0;
END_IF
END_METHOD

METHOD PROTECTED Initialize : BOOL
VAR_INPUT END_VAR
Initialize := SUPER^.Initialize();
END_METHOD

END_FUNCTION_BLOCK

